# B&R Automation Studio project Nitto (part 5)

#### CSV_ReadFile.ab
```automation-basic
FUNCTION_BLOCK CSV_ReadFile
;*****************************************************************
;FUB: 			CSV_ReadFile
;*****************************************************************
;Discription:
;	This FUB reads the Values from a CSV-File.
;
;Parameter:
;
;Author:	Georg Kreil
;			B&R Eggelsberg
;
;History:	V0.01 - 23 June 2003
;					created
;			V0.01.1 - 4 July 2003
;					no changes
;			V0.01.2 - 8 July 2003
;					Error with array-structures corrected
;			V0.01.3 - 14 July 2003
;					Error with array-structures corrected
;			V0.01.4 - 15 July 2003
;					Error by empty rows corrected
;			V0.01.5 - 17 July 2003
;					Error, when variable starts with array-structure, corrected
;			V0.01.6 - 21 July 2003
;					strings can have all possible character without ";"
;			V0.01.7 - 7 August 2003
;					no changes
;			V0.01.8 - 8 August 2003
;					no changes
;			V0.01.9 - 11 August 2003
;					Value error corrected
;			V0.02.0
;					no changes
;			V0.02.1
;					no changes
;			V0.02.2 - 11 August 2003
;					Datatypcontrol enable/disable
;			V0.02.3
;					no changes
;			V0.02.4 - 4 November 2003
;					Datatyperror in loop corrected
;			V0.02.5 - 13 November 2003
;					Real values error corrected (5e-7)
;			V0.02.6 - 14 November 2003
;					dynamic varible now possible
;			V0.02.7 - 24 November 2003
;					bugfixes
;			V0.02.8 - 27 November 2003
;					changing 80 characters per cyclic to one row per cyclic
;					different bugfixes
;			V0.03.1 - 21 January 2004
;					using the created strings from FUB CSV_ListFile with date
;			V0.03.3 - 12 May 2004
;					array behind array-structure corrected
;			V0.03.4 - 14 May 2004
;					changed the UDINT-conversion from STRING (see CSV_SEARCH)
;					corrected the STRING-datatypcontrol (1Byte error)
;			V0.03.9 - 2 August 2004
;					correction "only array" and "only array in struct"
;
;*****************************************************************
temp_status = temp_status
Options = Options

Internal.CharPerCyclic= 80		; number of character

loop Internal.y=0 to 10 do
	select Internal.Step

		;##########################################################################################
		state WAIT
		;##########################################################################################

			Internal.FileIdent= 0
			Internal.temp_status=0
			VarCnt = 0
			Internal.Separator = Separator

			if( (Internal.Separator = '.') or (Internal.Separator = '[') or (Internal.Separator = ']') or (Internal.Separator <= 32) or ( (Internal.Separator >= '0') and (Internal.Separator <= '9') ) or ( (Internal.Separator >= 'a') and (Internal.Separator <= 'z') ) or ( (Internal.Separator >= 'A') and (Internal.Separator <= 'Z') ) ) then
				status = ERROR_WRONG_SEPARATOR
				exitif(1=1)
			endif

			strcpy(adr(Internal.FileName),pFileName)
			if (Internal.y=0) then
				if( strlen(adr(Internal.FileName)) <> 0 ) then
					; control, if the filename has the right extension
					loop Internal.i=0 to sizeof(Internal.FileName) do

						Dyn_Usint access (adr(Internal.FileName)+Internal.i)

						; this is for using the created strings from FUB CSV_ListFile
						if (Dyn_Usint = ' ') then
							Dyn_Usint= 0
							; add extension to filename
							strcpy((adr(Internal.FileName)+Internal.i),".CSV")
							exitif(1=1)
						endif

						if(Dyn_Usint = '.')then
							if ( strcmp((adr(Internal.FileName)+Internal.i),".CSV") = 0 ) or ( strcmp((adr(Internal.FileName)+Internal.i),".csv") = 0 ) then
								exitif(1=1)
							else
								; replace wrong extension
								strcpy((adr(Internal.FileName)+Internal.i),".CSV")
								exitif(1=1)
							endif
						else if(Dyn_Usint = 0) then
							; add extension to filename
							strcpy((adr(Internal.FileName)+Internal.i),".CSV")
							exitif(1=1)
						endif

					endloop
					Internal.ArrayStructureStarts= 0
					status= 65535
					;Pathname angegeben
					if(pPath <> 0)then
						strcpy(adr(Internal.Path),pPath)
						; Pathname bearbeiten
						if( strlen(adr(Internal.Path)) <> 0 )then

						; control, if the filename has the right extension
							loop Internal.i=0 to sizeof(Internal.Path) do

								Dyn_Usint access (adr(Internal.Path) + Internal.i)
								 if( ((Dyn_Usint >= '0' ) and ( Dyn_Usint <= '9' )) or ((Dyn_Usint >= 'A') and (Dyn_Usint <= 'Z')) or ((Dyn_Usint >= 'a') and (Dyn_Usint <= 'z')) or ( Dyn_Usint = '_') or ( Dyn_Usint = '-') or ( Dyn_Usint = '/') or ( Dyn_Usint = '\') or ( Dyn_Usint = 0) )then

									if(Dyn_Usint = 0) then
										Dyn_Usint access (adr(Internal.Path) + Internal.i - 1)
										if(Dyn_Usint <> '\') and (Dyn_Usint <> '/')then
											strcat( adr(Internal.Path), adr("/") )
										endif
										exitif(1=1)
									endif
									status= 65535
								else
									status= INVALID_CHARACTER
									exitif(1=1)
								endif
							endloop
							strcat( adr(Internal.Path), adr(Internal.FileName) )
							strcpy( adr(Internal.FileName), adr(Internal.Path) )
						endif
					endif

				else
					status= NO_FILENAME
				endif
			endif

			when (1=1) and (Internal.y=0) do
			next FILE_OPEN

		;##########################################################################################
		state FILE_OPEN
		;##########################################################################################

			FileOpen_CSV.enable= 1
			FileOpen_CSV.pDevice= pDevice
			FileOpen_CSV.pFile= adr(Internal.FileName)
			FileOpen_CSV.mode= 2	;FILE_RW
			FileOpen_CSV FUB FileOpen()

			; no error
			when (FileOpen_CSV.status = 0) do
				Internal.FileIdent= FileOpen_CSV.ident
				; allocate memory, to copy the whole file
				Internal.status_alloc= TMP_alloc(FileOpen_CSV.filelen,adr(Internal.pFileData))
				strcpy(adr(Internal.FileName),"")
				status= 65535
			next FILE_READ

			; file is opening
			when (FileOpen_CSV.status = 65535) do
				status= FileOpen_CSV.status
			next FILE_OPEN

			;error durring
			when (FileOpen_CSV.status <> 0) and (FileOpen_CSV.status <> 65535) do
				status= FileOpen_CSV.status
			next WAIT

		;##########################################################################################
		state FILE_READ
		;##########################################################################################

			if( (Internal.status_alloc = 0) and (FileOpen_CSV.status = 0) )then
				FileRead_CSV.enable= 1
				FileRead_CSV.ident= Internal.FileIdent
				FileRead_CSV.offset= 0
				FileRead_CSV.pDest= Internal.pFileData
				FileRead_CSV.len= FileOpen_CSV.filelen
				FileRead_CSV FUB FileRead()
			endif

			when  (Internal.status_alloc <> 0) do
				status= Internal.status_alloc
			next WAIT

			when (FileRead_CSV.status <> 0) and  (FileRead_CSV.status <> 65535) do
				status= FileRead_CSV.status
			next WAIT

			when (FileRead_CSV.status = 65535) do
				status= FileRead_CSV.status
			next FILE_READ

			when (FileRead_CSV.status = 0) do
				Internal.Offset= 0
				Internal.OffsetOld= 0
				Internal.i= 0
				strcpy(adr(Internal.Value),"")
				strcpy(adr(Internal.TmpName),"")
				strcpy(adr(Internal.StructName),"")
				strcpy(adr(Internal.DataTyp),"")
				strcpy(adr(Internal.DateTime),"")
				strcpy(adr(Internal.VarName),"")
				Internal.OnlyArray= 0
				Internal.OnlyArrayInStruct= 0
				LineCnt= 0
				status= 65535
				ErrorNumber = 0
				ErrorLine = 0
				ErrorCnt = 0
			next FILE_CLOSE

		;##########################################################################################
		state FILE_CLOSE
		;##########################################################################################

		 	FileClose_CSV.enable= 1
			FileClose_CSV.ident= Internal.FileIdent
			FileClose_CSV FUB FileClose()

			; Fehler beim Schliessen
			when (FileClose_CSV.status <> 0) and (FileClose_CSV.status <> 65535) do
				status= FileClose_CSV.status
			next WAIT

			; kein Fehler aufgetreten
			when (FileClose_CSV.status = 0) do
				status= 65535
			next SEARCH_STRUCT_NAME

			; noch nicht fertig
			when (FileClose_CSV.status = 65535) do
				status= FileClose_CSV.status
			next FILE_CLOSE

		;##########################################################################################
		state SEARCH_STRUCT_NAME
		;##########################################################################################

		when (Internal.Offset >= FileOpen_CSV.filelen) or (status <> 65535) do
		next TEMP_FREE

		loop
			SearchChar access Internal.pFileData + Internal.Offset
			TestUsint = SearchChar

			if( SearchChar = 13 )then
				LineCnt= LineCnt+1
			endif

			if( SearchChar = '/' ) and (Internal.NameEntered <> 2) then
				Internal.HeaderLine= 1
			; date and time
			else if( (((SearchChar >= '0' ) and ( SearchChar <= '9' )) or ((SearchChar >= 'A') and (SearchChar <= 'Z')) or ((SearchChar >= 'a') and (SearchChar <= 'z')) or ( SearchChar = '.') or (SearchChar = ':') or (SearchChar = ' ') ) and (strcmp(adr(Internal.DataTyp),"DATE_AND_TIME") = 0 ) and (Internal.NameEntered = 2) and (Internal.HeaderLine = 0) )then			; neue Zeile
				Internal.DateTime[Internal.j]= SearchChar
				Internal.j= Internal.j+1
				Internal.DateAndTime= 1
			; only numbers
			else if( (((SearchChar >= '0' ) and ( SearchChar <= '9' )) or ( SearchChar = '.')  or ( SearchChar = 'E') or ( SearchChar = 'e') or ( SearchChar = '-')) and (Internal.NameEntered = 2) and (Internal.HeaderLine = 0) )then			; neue Zeile
				Internal.Value[Internal.j]= SearchChar
				Internal.j= Internal.j+1
			; Strings
	;		else if( (((SearchChar >= '0' ) and ( SearchChar <= '9' )) or ((SearchChar >= 'A') and (SearchChar <= 'Z')) or((SearchChar >= 'a') and (SearchChar <= 'z'))  or ( SearchChar = '.') or ( SearchChar = ' ')) and (Internal.NameEntered = 2) and (strcmp(adr(Internal.DataTyp),"STRING") = 0) and (Internal.HeaderLine = 0) )then			; neue Zeile
	;		else if( (((SearchChar >= 33 ) and ( SearchChar <= 58 )) or ((SearchChar >= 60 ) and ( SearchChar <= 126 )) or ( SearchChar = ' ') ) and (Internal.NameEntered = 2) and (strcmp(adr(Internal.DataTyp),"STRING") = 0) and (Internal.HeaderLine = 0) )then			; neue Zeile
;			alle sinnvollen Zeichen zulassen, auch Sonderzeichen
			else if( (SearchChar >= 32 ) and ( SearchChar <= 126 ) and (Internal.NameEntered = 2) and (strcmp(adr(Internal.DataTyp),"STRING") = 0) and (Internal.HeaderLine = 0) )then			; neue Zeile
				Internal.Value[Internal.j]= SearchChar
				Internal.j= Internal.j+1
			else if( ((SearchChar >= 'A') and (SearchChar <= 'Z')) or ((SearchChar >= 'a') and (SearchChar <= 'z')) or ((SearchChar >= '0' ) and ( SearchChar <= '9' )) or (SearchChar = '.') or (SearchChar = ':') or (SearchChar = '*') or (SearchChar = '[') or (SearchChar = ']') or (SearchChar = '_') and (Internal.HeaderLine = 0) )then
				Internal.TmpName[Internal.i]= SearchChar
				Internal.i= Internal.i+1
			else if( SearchChar = 13 ) or ( SearchChar = 10 )  then			; neue Zeile
				SearchChar access Internal.pFileData + Internal.Offset+1
				TestUsint = SearchChar
				if( SearchChar = 10) or ( SearchChar = 13 ) then
	;				LineCnt= LineCnt+1
					if(Internal.NameEntered = 1) then
						Internal.TmpName[Internal.i]= 0
						Internal.i= 0
						strcpy(adr(Internal.DataTyp),adr(Internal.TmpName))
					endif
					Internal.Value[Internal.j]= 0
					Internal.DateTime[Internal.j]= 0
					Internal.i= 0
					Internal.j= 0
					Internal.TmpName[Internal.i]= 0
					Internal.NameEntered= 0
					Internal.HeaderLine= 0
					inc(Internal.Offset)
					exitif(strlen(adr(Internal.StructName)) <> 0)
	;				exitif(1=1)
				else
	;				LineCnt= LineCnt+1
					if(Internal.NameEntered = 1) then
						Internal.TmpName[Internal.i]= 0
						Internal.i= 0
						strcpy(adr(Internal.DataTyp),adr(Internal.TmpName))
					endif
					Internal.Value[Internal.j]= 0
					Internal.DateTime[Internal.j]= 0
					Internal.i= 0
					Internal.j= 0
					Internal.TmpName[Internal.i]= 0
					Internal.NameEntered= 0
					Internal.HeaderLine= 0
					exitif(strlen(adr(Internal.StructName)) <> 0)
	;				exitif(1=1)
				endif
			; the structure name was readed
			else if( SearchChar = Internal.Separator) and (Internal.NameEntered = 0) and (Internal.HeaderLine = 0) then		; neuer Name
				Internal.TmpName[Internal.i]= 0
				Internal.i= 0
				strcpy(adr(Internal.StructName),adr(Internal.TmpName))
				Internal.NameEntered= 1
			; dataype was readed
			else if( SearchChar = Internal.Separator) and (Internal.NameEntered = 1) and (Internal.HeaderLine = 0) then		; neuer Datentyp
				Internal.TmpName[Internal.i]= 0
				Internal.i= 0
				strcpy(adr(Internal.DataTyp),adr(Internal.TmpName))
				Internal.NameEntered= 2
			; value was readed
			else if( SearchChar = Internal.Separator) and (Internal.NameEntered = 2) and (Internal.HeaderLine = 0) then		; weitere Spalten ignorieren
				Internal.TmpName[Internal.j]= 0
				Internal.NameEntered= 3

			else if( SearchChar = ' ') and (Internal.NameEntered = 0) and (Internal.HeaderLine = 0) then		; Leerzeichen
				Internal.SpacesCounter= Internal.SpacesCounter+1
			endif
			exitif(Internal.Offset >= FileOpen_CSV.filelen+1)
			inc(Internal.Offset)
		endloop

		Internal.Offset= Internal.Offset+1
		Internal.OffsetOld= Internal.Offset
		memcpy(adr(Internal.TmpDataTyp),adr(Internal.DataTyp),5)
		Internal.TmpDataTyp[5]= 0

;		when (RowNotOnEnd = 1) do
;			status= 65535
;		next SEARCH_STRUCT_NAME

		; is it a dynamic variable
		if(Internal.StructName[0] = '*')then
			Internal.DynamicVariable= 1
		else
			Internal.DynamicVariable= 0
		endif

		;######################################################
		; Correction 15.July 2003
		when ( strlen(adr(Internal.StructName)) = 0  )do
			status= 65535
		next SEARCH_STRUCT_NAME
		; Correction 15.July 2003
		;######################################################

		when (Internal.HeaderLine = 1)do
			status= 65535
		next SEARCH_STRUCT_NAME

		;######################################################
		; Correction 17.July 2003
		when( strcmp(adr(Internal.DataTyp),"ARRAY_OF_STRUCTURES") = 0 ) do
			loop Internal.i=strlen(adr(Internal.StructName)) downto 0 do	;Kommastellen löschen
				SearchChar access adr(Internal.StructName)+Internal.i
				if(SearchChar ='.')then
					SearchChar= 0
					Part=1
					exitif(1=1)
				endif
			endloop
			if(	Part = 0 )then
				Internal.ArrayStructureStarts= 1
				strcpy(adr(Internal.StructName),"")
				Internal.i= 0
				Internal.SpacesCounter= 0
			else
				strcat(adr(Internal.StructName),adr(Internal.VarName))
				Internal.i= 0
				Internal.SpacesCounter= 0
				Part= 0
				status= 65535
			endif
		next SEARCH_VAR_NAMES

	;	when( ( strcmp(adr(Internal.DataTyp),"STRUCTURE") = 0 ) or ( strcmp(adr(Internal.DataTyp),"ARRAY_OF_STRUCTURES") = 0 ) ) do
		when ( strcmp(adr(Internal.DataTyp),"STRUCTURE") = 0 ) do
		; Correction 17.July 2003
		;######################################################
			Internal.level= 2
			loop Internal.i=0 to strlen(adr(Internal.StructName)) do
				SearchChar access adr(Internal.StructName)+Internal.i
				if(SearchChar ='.') and( Internal.level = ((Internal.SpacesCounter+1)/5) ) then
					SearchChar= 0
					exitif(1=1)
				else if(SearchChar =']') and( Internal.level = ((Internal.SpacesCounter+1)/5) ) then
					SearchChar access adr(Internal.StructName)+Internal.Merker
					SearchChar= 0
					exitif(1=1)
				else if (SearchChar ='.') and ( Internal.level < ((Internal.SpacesCounter+1)/5) ) then
					Internal.level= Internal.level+1
				else if (SearchChar =']') and ( Internal.level < ((Internal.SpacesCounter+1)/5) ) then
					Internal.level= Internal.level+1
				endif
			endloop
			Internal.i=0

			strcat(adr(Internal.StructName),adr(Internal.VarName))

			Internal.SpacesCounter= 0
			status= 65535
		next SEARCH_VAR_NAMES

		when(strcmp(adr(Internal.TmpDataTyp),"ARRAY") = 0 ) do
			Internal.OnlyArray= 1
			loop Internal.i=strlen(adr(Internal.StructName)) downto 0 do
				SearchChar access adr(Internal.StructName) + Internal.i
				if(SearchChar ='.')then
					SearchChar = 0
					Internal.OnlyArray= 0
					Internal.OnlyArrayInStruct= 1
					exitif(1=1)
				endif
			endloop

			Internal.i=0
			status= 65535
		next SEARCH_VAR_NAMES

		when( 1=1 ) do
			Internal.level= 2
			loop Internal.i=0 to strlen(adr(Internal.StructName)) do
				SearchChar access adr(Internal.StructName)+Internal.i
				if(SearchChar ='.') and( Internal.level = ((Internal.SpacesCounter+1)/5) ) then
					SearchChar= 0
					exitif(1=1)
				else if(SearchChar =']') and( Internal.level = ((Internal.SpacesCounter+1)/5) ) then
					SearchChar access adr(Internal.StructName)+Internal.Merker
					SearchChar= 0
					exitif(1=1)
				else if (SearchChar ='.') and ( Internal.level < ((Internal.SpacesCounter+1)/5) ) then
					Internal.level= Internal.level+1
				else if (SearchChar =']') and ( Internal.level < ((Internal.SpacesCounter+1)/5) ) then
					Internal.level= Internal.level+1
				endif
			endloop
			Internal.i=0
			strcat(adr(Internal.StructName),adr(Internal.VarName))

			Internal.SpacesCounter= 0
			status= 65535
		next SET_VARIABLE

		;##########################################################################################
		state SEARCH_VAR_NAMES
		;##########################################################################################

		when (Internal.Offset >= FileOpen_CSV.filelen) or (status <> 65535) do
		next TEMP_FREE

		loop
			SearchChar access Internal.pFileData + Internal.Offset
			TestUsint = SearchChar

			if( LineCnt = 64 )then
				LineCnt = LineCnt
			endif

			if( SearchChar = 13 )then
				LineCnt= LineCnt+1
			endif

			if( SearchChar = '/' ) and (Internal.NameEntered <> 2) then
				Internal.HeaderLine= 1
			; Zeit/Datum
			else if( (((SearchChar >= '0' ) and ( SearchChar <= '9' )) or ((SearchChar >= 'A') and (SearchChar <= 'Z')) or ((SearchChar >= 'a') and (SearchChar <= 'z')) or ( SearchChar = '.') or (SearchChar = ':') or (SearchChar = ' ') ) and (strcmp(adr(Internal.DataTyp),"DATE_AND_TIME") = 0 ) and (Internal.NameEntered = 2) and (Internal.HeaderLine = 0)  )then			; neue Zeile
				Internal.DateTime[Internal.j]= SearchChar
				Internal.j= Internal.j+1
			; Nur Zahlenwert
			else if( (((SearchChar >= '0' ) and ( SearchChar <= '9' )) or ( SearchChar = '.')  or ( SearchChar = 'E') or ( SearchChar = 'e') or ( SearchChar = '-')) and (Internal.NameEntered = 2) and (Internal.HeaderLine = 0) )then			; neue Zeile
				Internal.Value[Internal.j]= SearchChar
				Internal.j= Internal.j+1
			; String-Wert
	;		else if( (((SearchChar >= '0' ) and ( SearchChar <= '9' )) or ((SearchChar >= 'A') and (SearchChar <= 'Z')) or((SearchChar >= 'a') and (SearchChar <= 'z'))  or ( SearchChar = '.') or ( SearchChar = ' ')) and (Internal.NameEntered = 2) and (strcmp(adr(Internal.DataTyp),"STRING") = 0) and (Internal.HeaderLine = 0) )then			; neue Zeile
;			else if( (((SearchChar >= 33 ) and ( SearchChar <= 58 )) or ((SearchChar >= 60 ) and ( SearchChar <= 126 )) or ( SearchChar = ' ') ) and (Internal.NameEntered = 2) and (strcmp(adr(Internal.DataTyp),"STRING") = 0) and (Internal.HeaderLine = 0) )then			; neue Zeile
;			alle sinnvollen Zeichen zulassen, auch Sonderzeichen
			else if( (SearchChar >= 32 ) and ( SearchChar <= 126 ) and (Internal.NameEntered = 2) and (strcmp(adr(Internal.DataTyp),"STRING") = 0) and (Internal.HeaderLine = 0) )then			; neue Zeile
				Internal.Value[Internal.j]= SearchChar
				Internal.j= Internal.j+1
			else if( ((SearchChar >= 'A') and (SearchChar <= 'Z')) or ((SearchChar >= 'a') and (SearchChar <= 'z')) or ((SearchChar >= '0' ) and ( SearchChar <= '9' )) or (SearchChar = '.') or (SearchChar = ':') or (SearchChar = '*') or (SearchChar = '[') or (SearchChar = ']') or (SearchChar = '_') and (Internal.HeaderLine = 0) )then
				Internal.TmpName[Internal.i]= SearchChar
				Internal.i= Internal.i+1
			else if( SearchChar = 13 ) or ( SearchChar = 10 )  then			; neue Zeile
				Internal.Offset= Internal.Offset+1
	;			LineCnt= LineCnt+1
				SearchChar access Internal.pFileData + Internal.Offset
				TestUsint = SearchChar
				if( SearchChar = 10) or ( SearchChar = 13 ) then
	;				LineCnt= LineCnt+1
					if(Internal.NameEntered = 1) then
						Internal.TmpName[Internal.i]= 0
						Internal.i= 0
						strcpy(adr(Internal.DataTyp),adr(Internal.TmpName))
					endif
					Internal.Value[Internal.j]= 0
					Internal.DateTime[Internal.j]= 0
					Internal.i= 0
					Internal.j= 0
					Internal.TmpName[Internal.i]= 0
					Internal.NameEntered= 0
					inc(Internal.Offset)
;					Internal.HeaderLine= 0
					exitif( (strlen(adr(Internal.VarName)) <> 0) or (Internal.HeaderLine= 1) )
				else
	;				LineCnt= LineCnt+1
					if(Internal.NameEntered = 1) then
						Internal.TmpName[Internal.i]= 0
						Internal.i= 0
						strcpy(adr(Internal.DataTyp),adr(Internal.TmpName))
					endif
					if(strlen(adr(Internal.VarName)) = 0) then
						Internal.Offset= Internal.Offset-1
					endif
					Internal.Value[Internal.j]= 0
					Internal.DateTime[Internal.j]= 0
					Internal.i= 0
					Internal.j= 0
					Internal.TmpName[Internal.i]= 0
					Internal.NameEntered= 0
;					Internal.HeaderLine= 0
					exitif( (strlen(adr(Internal.VarName)) <> 0) or (Internal.HeaderLine= 1) )
				endif
			; Strukturname
			else if( SearchChar = Internal.Separator) and (Internal.NameEntered = 0) and (Internal.HeaderLine = 0) then		; neuer Name
				Internal.TmpName[Internal.i]= 0
				Internal.i= 0
				Internal.j= 0			; Correction 11 August 2003
				strcpy(adr(Internal.VarName),adr(Internal.TmpName))
				Internal.NameEntered= 1
			; Datenyp
			else if( SearchChar = Internal.Separator) and (Internal.NameEntered = 1) and (Internal.HeaderLine = 0) then		; neuer Datentyp
				Internal.TmpName[Internal.i]= 0
				Internal.i= 0
				Internal.j= 0			; Correction 11 August 2003
				strcpy(adr(Internal.DataTyp),adr(Internal.TmpName))
				Internal.NameEntered= 2

			else if( SearchChar = Internal.Separator) and (Internal.NameEntered = 2) and (Internal.HeaderLine = 0) then		; weitere Spalten ignorieren
				Internal.TmpName[Internal.j]= 0
				Internal.NameEntered= 3

			else if( SearchChar = ' ') and (Internal.NameEntered = 0) and (Internal.HeaderLine = 0) then		; Leerzeichen
				Internal.SpacesCounter= Internal.SpacesCounter+1
			endif
			exitif(Internal.Offset >= FileOpen_CSV.filelen+1)
			inc(Internal.Offset)
		endloop

	;	Internal.Offset= Internal.Offset+1
			Internal.Offset= Internal.Offset
		Internal.OffsetOld= Internal.Offset
		memcpy(adr(Internal.TmpDataTyp),adr(Internal.DataTyp),5)
		Internal.TmpDataTyp[5]= 0

;		when (RowNotOnEnd = 1) do
;			status= 65535
;		next SEARCH_VAR_NAMES

		when (Internal.HeaderLine = 1)do
			Internal.HeaderLine = 0
			Internal.i= 0
			strcpy(adr(Internal.Value),"")
			strcpy(adr(Internal.TmpName),"")
			strcpy(adr(Internal.StructName),"")
			strcpy(adr(Internal.DataTyp),"")
			strcpy(adr(Internal.DateTime),"")
			strcpy(adr(Internal.VarName),"")
			Internal.OnlyArray= 0
			Internal.OnlyArrayInStruct= 0
			Internal.ArrayStructureStarts = 0
			status= 65535
		next SEARCH_STRUCT_NAME

		;######################################################
		; Correction 6.October 2003
		when ( strlen(adr(Internal.StructName)) = 0  )and (Internal.ArrayStructureStarts = 0) do
			status= 65535
		next SEARCH_STRUCT_NAME
		; Correction 6.October 2003
		;######################################################

		;no new variablename in csv-file found
		when (Internal.VarName[0] = 0) do
			Internal.StructName[0]= 0
			status= 65535
		next SEARCH_STRUCT_NAME

		; full name found
		when(Internal.VarName[0]<> '.') do
			strcpy(adr(Internal.StructName),adr(Internal.VarName))
			status= 65535
		next SET_VARIABLE

		; only array-variable -> no structure, no single variable
		when(Internal.OnlyArray = 1) do
			; is it a dynamic variable
			if(Internal.DynamicVariable = 1)then
				strcat( adr(Internal.StructName), "*" )
				strcat( adr(Internal.StructName), adr(Internal.VarName)+1)
			else
				strcpy( adr(Internal.StructName), adr(Internal.VarName)+1)
			endif

			status= 65535
		next SET_VARIABLE

		; only an array-variable in a structure -> no structure, no single variable
		when(Internal.OnlyArrayInStruct = 1) do
			Internal.i=0
			strcat( adr(Internal.StructName), adr(Internal.VarName))
			status= 65535
		next SET_VARIABLE

		; beginn of an array of structures found
		when( strcmp(adr(Internal.DataTyp),"ARRAY_OF_STRUCTURES") = 0 ) do

			Internal.level= 2
			loop Internal.i=0 to strlen(adr(Internal.StructName)) do
				SearchChar access adr(Internal.StructName)+Internal.i
				if(SearchChar ='.') and( Internal.level = ((Internal.SpacesCounter+1)/5) ) then
					SearchChar= 0
					exitif(1=1)
				else if(SearchChar =']') and( Internal.level = ((Internal.SpacesCounter+1)/5) ) then
					SearchChar access adr(Internal.StructName)+Internal.Merker
					SearchChar= 0
					exitif(1=1)
				else if (SearchChar ='.') and ( Internal.level < ((Internal.SpacesCounter+1)/5) ) then
					Internal.level= Internal.level+1
				else if (SearchChar =']') and ( Internal.level < ((Internal.SpacesCounter+1)/5) ) then
					Internal.level= Internal.level+1
				endif
			endloop
			Internal.i=0
			Internal.SpacesCounter= 0
			status= 65535
		next SEARCH_VAR_NAMES

		;new array found
		when ( strcmp(adr(Internal.TmpDataTyp),"ARRAY") = 0 )do
			Internal.level= 2
			loop Internal.i=0 to strlen(adr(Internal.StructName)) do
				SearchChar access adr(Internal.StructName)+Internal.i
				if(SearchChar ='.') and( Internal.level = ((Internal.SpacesCounter+1)/5) ) then
					SearchChar= 0
					exitif(1=1)
				else if(SearchChar =']') and( Internal.level = ((Internal.SpacesCounter+1)/5) ) then
					SearchChar access adr(Internal.StructName)+Internal.Merker
					SearchChar= 0
					exitif(1=1)
				else if (SearchChar ='.') and ( Internal.level < ((Internal.SpacesCounter+1)/5) ) then
					Internal.level= Internal.level+1
				else if (SearchChar =']') and ( Internal.level < ((Internal.SpacesCounter+1)/5) ) then
					Internal.level= Internal.level+1
				endif
			endloop
			Internal.i=0
			Internal.SpacesLastRow= Internal.SpacesCounter
			Internal.SpacesCounter= 0
			status= 65535
		next SEARCH_VAR_NAMES

		; new structure found
		when( strcmp(adr(Internal.DataTyp),"STRUCTURE") = 0 ) do
		;######################################################
		; Correction 17.July 2003
			if (Internal.ArrayStructureStarts = 0) then
				Internal.level= 2
				loop Internal.i=0 to strlen(adr(Internal.StructName)) do
					SearchChar access adr(Internal.StructName)+Internal.i
					if(SearchChar ='.') and( Internal.level = ((Internal.SpacesCounter+1)/5) ) then
						SearchChar= 0
						exitif(1=1)
					else if(SearchChar =']') and( Internal.level = ((Internal.SpacesCounter+1)/5) ) then

						loop Internal.j=Internal.i downto 0 do
							SearchChar access adr(Internal.StructName)+Internal.j
							exitif(SearchChar = '.')
						endloop
						SearchChar= 0
						exitif(1=1)
					else if (SearchChar ='.') and ( Internal.level < ((Internal.SpacesCounter+1)/5) ) then
						Internal.level= Internal.level+1
					else if (SearchChar =']') and ( Internal.level < ((Internal.SpacesCounter+1)/5) ) then
						Internal.level= Internal.level+1
					endif
				endloop
				Internal.i=0
				strcat(adr(Internal.StructName),adr(Internal.VarName))
			else
				Internal.level= 2
				if(( Internal.level <> ((Internal.SpacesCounter+1)/5) )) then
					loop Internal.i=0 to strlen(adr(Internal.StructName)) do
						SearchChar access adr(Internal.StructName)+Internal.i
						if(SearchChar ='.') and( Internal.level = ((Internal.SpacesCounter+1)/5) ) then
							SearchChar= 0
							exitif(1=1)
						else if(SearchChar =']') and( Internal.level = ((Internal.SpacesCounter+1)/5) ) then

							loop Internal.j=Internal.i downto 0 do
								SearchChar access adr(Internal.StructName)+Internal.j
								exitif(SearchChar = '.')
							endloop
							SearchChar= 0
							exitif(1=1)
						else if (SearchChar ='.') and ( Internal.level < ((Internal.SpacesCounter+1)/5) ) then
							Internal.level= Internal.level+1
						else if (SearchChar =']') and ( Internal.level < ((Internal.SpacesCounter+1)/5) ) then
							Internal.level= Internal.level+1
						endif
					endloop
				else
					Internal.i= 0
					; is it a dynamic variable
					if(Internal.DynamicVariable = 1)then
						strcpy( adr(Internal.StructName),"*" )
					else
						strcpy( adr(Internal.StructName),"" )
					endif
				endif

				if ( Internal.i = 0 ) then
					strcat(adr(Internal.StructName),adr(Internal.VarName)+1)
				else
					strcat(adr(Internal.StructName),adr(Internal.VarName))
				endif
				Internal.i=0
			endif
		; Correction 17.July 2003
		;######################################################

			Internal.SpacesCounter= 0
			status= 65535
		next SEARCH_VAR_NAMES

		when( 1=1 ) do
			Internal.level= 2
			loop Internal.i=0 to strlen(adr(Internal.StructName)) do
				SearchChar access adr(Internal.StructName)+Internal.i
				if(SearchChar ='.') and( Internal.level = ((Internal.SpacesCounter+1)/5) ) then
					SearchChar= 0
					exitif(1=1)
				else if(SearchChar =']') and( Internal.level = ((Internal.SpacesCounter+1)/5) ) then
					SearchChar access adr(Internal.StructName)+Internal.Merker
					SearchChar= 0
					exitif(1=1)
				else if (SearchChar ='.') and ( Internal.level < ((Internal.SpacesCounter+1)/5) ) then
					Internal.Merker= Internal.i
					Internal.level= Internal.level+1
				else if (SearchChar =']') and ( Internal.level < ((Internal.SpacesCounter+1)/5) ) then
					Internal.level= Internal.level+1
				endif
			endloop
			Internal.i=0
			strcat(adr(Internal.StructName),adr(Internal.VarName))

			Internal.SpacesCounter= 0
			status= 65535
		next SET_VARIABLE

		;##########################################################################################
		state SET_VARIABLE
		;##########################################################################################

		Internal.PV_xgetadrStatus= PV_xgetadr(adr(Internal.StructName), adr(Internal.PV_Adress), adr(Internal.data_len))
		Internal.PV_nInfoStatus= PV_ninfo(adr(Internal.StructName),adr(Internal.PVdata_typ),adr(Internal.datatyp_len),adr(Internal.dimension))

		when(	Internal.PV_xgetadrStatus <> 0 ) and (IgnoreError = FALSE) do
			Internal.OnlyArrayInStruct = 0
			if( ErrorNumber = 0 ) then
				ErrorNumber = Internal.PV_xgetadrStatus
				ErrorLine = LineCnt
			endif

			inc( ErrorCnt )
			status= Internal.PV_xgetadrStatus
		next TEMP_FREE

		when(	Internal.PV_xgetadrStatus <> 0 ) and (IgnoreError = TRUE) do
			if( ErrorNumber = 0 ) then
				ErrorNumber = Internal.PV_xgetadrStatus
				ErrorLine = LineCnt
			endif

			inc( ErrorCnt )

			status= 65535
		next SEARCH_VAR_NAMES

		Inc(VarCnt)

		if( (strcmp(adr(Internal.DataTyp),"BOOL") = 0 ) and (Internal.data_len = 1) and (Internal.PV_xgetadrStatus = 0) and (Internal.PV_nInfoStatus = 0) )then

			if (Internal.PVdata_typ = 1) then
				Dyn_Bool access Internal.PV_Adress
				loop Internal.i=strlen(adr(Internal.Value)) downto 0 do	;Kommastellen löschen
					SearchChar access adr(Internal.Value)+Internal.i
					if(SearchChar ='.')then
						SearchChar= 0
						exitif(1=1)
					endif
				endloop
				Dyn_Bool= bool( atoi(adr(Internal.Value)) )
				status= 65535
			else
				Internal.OnlyArrayInStruct = 0
				Internal.temp_status= DATATYP_ERROR
			endif

		else if( (strcmp(adr(Internal.DataTyp),"USINT") = 0 ) and (Internal.data_len = 1) and (Internal.PV_xgetadrStatus = 0) and (Internal.PV_nInfoStatus = 0) )then

			if (Internal.PVdata_typ = 5) then
				Dyn_Usint access Internal.PV_Adress
				loop Internal.i=strlen(adr(Internal.Value)) downto 0 do	;Kommastellen löschen
					SearchChar access adr(Internal.Value)+Internal.i
					if(SearchChar ='.')then
						SearchChar= 0
						exitif(1=1)
					endif
				endloop
				Dyn_Usint= usint( atoi(adr(Internal.Value)) )
				status= 65535
			else
				Internal.OnlyArrayInStruct = 0
				Internal.temp_status= DATATYP_ERROR
			endif

		else if( (strcmp(adr(Internal.DataTyp),"SINT") = 0 ) and (Internal.data_len = 1) and (Internal.PV_xgetadrStatus = 0) and (Internal.PV_nInfoStatus = 0) )then

			if (Internal.PVdata_typ = 2) then
				Dyn_Sint access Internal.PV_Adress
				loop Internal.i=strlen(adr(Internal.Value)) downto 0 do	;Kommastellen löschen
					SearchChar access adr(Internal.Value)+Internal.i
					if(SearchChar ='.')then
						SearchChar= 0
						exitif(1=1)
					endif
				endloop
				Dyn_Sint= sint( atoi(adr(Internal.Value)) )
				status= 65535
			else
				Internal.OnlyArrayInStruct = 0
				Internal.temp_status= DATATYP_ERROR
			endif

		else if( (strcmp(adr(Internal.DataTyp),"UINT") = 0 ) and (Internal.data_len = 2) and (Internal.PV_xgetadrStatus = 0) and (Internal.PV_nInfoStatus = 0) )then

			if (Internal.PVdata_typ = 6) then
				Dyn_Uint access Internal.PV_Adress
				loop Internal.i=strlen(adr(Internal.Value)) downto 0 do	;Kommastellen löschen
					SearchChar access adr(Internal.Value)+Internal.i
					if(SearchChar ='.')then
						SearchChar= 0
						exitif(1=1)
					endif
				endloop
				Dyn_Uint= uint( atoi(adr(Internal.Value)) )
				status= 65535
			else
				Internal.OnlyArrayInStruct = 0
				Internal.temp_status= DATATYP_ERROR
			endif

		else if( (strcmp(adr(Internal.DataTyp),"INT") = 0 ) and (Internal.data_len = 2) and (Internal.PV_xgetadrStatus = 0) and (Internal.PV_nInfoStatus = 0) )then

			if (Internal.PVdata_typ = 3) then
				Dyn_Int access Internal.PV_Adress
				loop Internal.i=strlen(adr(Internal.Value)) downto 0 do	;Kommastellen löschen
					SearchChar access adr(Internal.Value)+Internal.i
					if(SearchChar ='.')then
						SearchChar= 0
						exitif(1=1)
					endif
				endloop
				Dyn_Int= int( atoi(adr(Internal.Value)) )
				status= 65535
			else
				Internal.OnlyArrayInStruct = 0
				Internal.temp_status= DATATYP_ERROR
			endif

		else if( (strcmp(adr(Internal.DataTyp),"UDINT") = 0 ) and (Internal.data_len = 4) and (Internal.PV_xgetadrStatus = 0) and (Internal.PV_nInfoStatus = 0) )then

			if (Internal.PVdata_typ = 7) then
				Dyn_Udint access Internal.PV_Adress
				loop Internal.i=strlen(adr(Internal.Value)) downto 0 do	;Kommastellen löschen
					SearchChar access adr(Internal.Value)+Internal.i
					if(SearchChar ='.')then
						SearchChar= 0
						exitif(1=1)
					endif
				endloop

				if (Internal.Value[0] <> '-') then
					Dyn_Udint = 0
					Internal.j = usint(strlen(adr(Internal.Value)))
					loop Internal.i=0 to Internal.j do

						Dyn_Udint = Dyn_Udint+(Internal.Value[Internal.i]-48)*udint(EXPT(10,strlen(adr(Internal.Value))-Internal.i-1))

					endloop
				else
					Dyn_Udint= udint( atoi(adr(Internal.Value)) )
				endif
				status= 65535
			else
				Internal.OnlyArrayInStruct = 0
				Internal.temp_status= DATATYP_ERROR
			endif

		else if( (strcmp(adr(Internal.DataTyp),"DINT") = 0 ) and (Internal.data_len = 4) and (Internal.PV_xgetadrStatus = 0) and (Internal.PV_nInfoStatus = 0) )then

			if (Internal.PVdata_typ = 4) then
				Dyn_Dint access Internal.PV_Adress
				loop Internal.i=strlen(adr(Internal.Value)) downto 0 do	;Kommastellen löschen
					SearchChar access adr(Internal.Value)+Internal.i
					if(SearchChar ='.')then
						SearchChar= 0
						exitif(1=1)
					endif
				endloop
				Dyn_Dint= atoi(adr(Internal.Value))
				status= 65535
			else
				Internal.OnlyArrayInStruct = 0
				Internal.temp_status= DATATYP_ERROR
			endif

		else if( (strcmp(adr(Internal.DataTyp),"STRING") = 0 ) and ((Internal.data_len-1) <= sizeof(Dyn_String)) and ((Internal.data_len-1) >= strlen(adr(Internal.Value))) and (Internal.PV_xgetadrStatus = 0) and (Internal.PV_nInfoStatus = 0) )then

			if (Internal.PVdata_typ = 9) then
				Dyn_String access Internal.PV_Adress
				strcpy(adr(Dyn_String),adr(Internal.Value))
				status= 65535
			else
				Internal.OnlyArrayInStruct = 0
				Internal.temp_status= DATATYP_ERROR
			endif

		else if( (strcmp(adr(Internal.DataTyp),"REAL") = 0 ) and (Internal.data_len = 4) and (Internal.PV_xgetadrStatus = 0) and (Internal.PV_nInfoStatus = 0) )then

			if (Internal.PVdata_typ = 8) then
				Dyn_Real access Internal.PV_Adress
				Dyn_Real= atof(adr(Internal.Value))
				status= 65535
			else
				Internal.OnlyArrayInStruct = 0
				Internal.temp_status= DATATYP_ERROR
			endif

		else if ((strcmp(adr(Internal.DataTyp),"LREAL") = 0 ) and (Internal.data_len = 8) and (Internal.PV_xgetadrStatus = 0) and (Internal.PV_nInfoStatus = 0) )then

			if (Internal.PVdata_typ = 14) then
				Dyn_LReal access Internal.PV_Adress
				Dyn_LReal= CSV_AtoDouble(adr(Internal.Value))
				status= 65535
			else
				Internal.OnlyArrayInStruct = 0
				Internal.temp_status= DATATYP_ERROR
			endif

		else if( (strcmp(adr(Internal.DataTyp),"OCTET STRING") = 0 ) and ((Internal.data_len-1) <= sizeof(Dyn_String)) and ((Internal.data_len-1) >= strlen(adr(Internal.Value))) and (Internal.PV_xgetadrStatus = 0) )then
			Dyn_String access Internal.PV_Adress
			strcpy(adr(Dyn_String),adr(Internal.Value))
			status= 65535

		else if( (strcmp(adr(Internal.DataTyp),"DATE_AND_TIME") = 0 ) and (Internal.data_len = 4) and (Internal.PV_xgetadrStatus = 0) and (Internal.PV_nInfoStatus = 0) )then

			if (Internal.PVdata_typ = 11) then
				Internal.Counter= 0
				loop Internal.i=0 to strlen(adr(Internal.DateTime)) do
					SearchChar access adr(Internal.DateTime)+Internal.i
					if( (SearchChar <> ' ') and (SearchChar <> ':') and (SearchChar <> 0) )then
						Internal.TmpDateTime[Internal.j]= SearchChar
						Internal.j= Internal.j+1
					else if( ((SearchChar = ' ') and (Internal.Counter < 3)) or ((SearchChar = ' ') and (Internal.Counter >= 5)) or ((SearchChar = ':') and (Internal.Counter >= 3)) or (SearchChar = 0) )then
						Internal.TmpDateTime[Internal.j]= 0
						; Tag
						if(Internal.Counter = 0) then
							if(strcmp(adr(Internal.TmpDateTime),"Sun") = 0 )then
								Internal.DateTimeStruct.wday= 0
								Internal.Counter = 1
							else if(strcmp(adr(Internal.TmpDateTime),"Mon") = 0 )then
								Internal.DateTimeStruct.wday= 1
								Internal.Counter = 1
							else if(strcmp(adr(Internal.TmpDateTime),"Tue") = 0 )then
								Internal.DateTimeStruct.wday= 2
								Internal.Counter = 1
							else if(strcmp(adr(Internal.TmpDateTime),"Wed") = 0 )then
								Internal.DateTimeStruct.wday= 3
								Internal.Counter = 1
							else if(strcmp(adr(Internal.TmpDateTime),"Thu") = 0 )then
								Internal.DateTimeStruct.wday= 4
								Internal.Counter = 1
							else if(strcmp(adr(Internal.TmpDateTime),"Fri") = 0 )then
								Internal.DateTimeStruct.wday= 5
								Internal.Counter = 1
							else if(strcmp(adr(Internal.TmpDateTime),"Sat") = 0 )then
								Internal.DateTimeStruct.wday= 6
								Internal.Counter = 1
							endif
						;Datum
						else if(Internal.Counter = 1) then
							if(strcmp(adr(Internal.TmpDateTime),"Jan") = 0 )then
								Internal.DateTimeStruct.month= 1
								Internal.Counter= 2
							else if(strcmp(adr(Internal.TmpDateTime),"Feb") = 0 )then
								Internal.DateTimeStruct.month= 2
								Internal.Counter= 2
							else if(strcmp(adr(Internal.TmpDateTime),"Mar") = 0 )then
								Internal.DateTimeStruct.month= 3
								Internal.Counter= 2
							else if(strcmp(adr(Internal.TmpDateTime),"Apr") = 0 )then
								Internal.DateTimeStruct.month= 4
								Internal.Counter= 2
							else if(strcmp(adr(Internal.TmpDateTime),"May") = 0 )then
								Internal.DateTimeStruct.month= 5
								Internal.Counter= 2
							else if(strcmp(adr(Internal.TmpDateTime),"Jun") = 0 )then
								Internal.DateTimeStruct.month= 6
								Internal.Counter= 2
							else if(strcmp(adr(Internal.TmpDateTime),"Jul") = 0 )then
								Internal.DateTimeStruct.month= 7
								Internal.Counter= 2
							else if(strcmp(adr(Internal.TmpDateTime),"Aug") = 0 )then
								Internal.DateTimeStruct.month= 8
								Internal.Counter= 2
							else if(strcmp(adr(Internal.TmpDateTime),"Sep") = 0 )then
								Internal.DateTimeStruct.month= 9
								Internal.Counter= 2
							else if(strcmp(adr(Internal.TmpDateTime),"Oct") = 0 )then
								Internal.DateTimeStruct.month= 10
								Internal.Counter= 2
							else if(strcmp(adr(Internal.TmpDateTime),"Nov") = 0 )then
								Internal.DateTimeStruct.month= 11
								Internal.Counter= 2
							else if(strcmp(adr(Internal.TmpDateTime),"Dec") = 0 )then
								Internal.DateTimeStruct.month= 12
								Internal.Counter= 2
							endif

						else if(Internal.Counter = 2) then
								Internal.DateTimeStruct.day= usint( atoi(adr(Internal.TmpDateTime)) )
								Internal.Counter= 3

						else if(Internal.Counter = 3) then
								Internal.DateTimeStruct.hour= usint( atoi(adr(Internal.TmpDateTime)) )
								Internal.Counter= 4

						else if(Internal.Counter = 4) then
								Internal.DateTimeStruct.minute= usint( atoi(adr(Internal.TmpDateTime)) )
								Internal.Counter= 5

						else if(Internal.Counter = 5) then
								Internal.DateTimeStruct.second= usint( atoi(adr(Internal.TmpDateTime)) )
								Internal.Counter= 6

						else if(Internal.Counter = 6) then
								Internal.DateTimeStruct.year= uint( atoi(adr(Internal.TmpDateTime)) )
								Internal.Counter= 7
						endif
						Internal.j= 0
					endif

				endloop
				Internal.i= 0
				Dyn_Date_and_Time access Internal.PV_Adress
				Dyn_Date_and_Time= DTStructure_TO_DT(adr(Internal.DateTimeStruct))
				Internal.DateAndTime = 0
				status= 65535
			else
				Internal.OnlyArrayInStruct = 0
				Internal.temp_status= DATATYP_ERROR
			endif

		else if( (strcmp(adr(Internal.DataTyp),"TIME") = 0 ) and (Internal.data_len = 4) and (Internal.PV_xgetadrStatus = 0) and (Internal.PV_nInfoStatus = 0) )then

			if (Internal.PVdata_typ = 12) then
				Dyn_Time access Internal.PV_Adress

				loop Internal.i=strlen(adr(Internal.Value)) downto 0 do	;Kommastellen löschen
					SearchChar access adr(Internal.Value)+Internal.i
					if(SearchChar ='.')then
						SearchChar= 0
						exitif(1=1)
					endif
				endloop
				Dyn_Time= time( atoi(adr(Internal.Value)) )
				status= 65535
			else
				Internal.OnlyArrayInStruct = 0
				Internal.temp_status= DATATYP_ERROR
			endif

		;######################################################################
		; keine DatentypKontrolle
		else if(No_DatatypControl = 1) and (Internal.PV_xgetadrStatus = 0) then
			; 1-Byte (BOOL,SINT,USINT)
			if (Internal.data_len = 1)	then
				Dyn_Usint access Internal.PV_Adress
				loop Internal.i=strlen(adr(Internal.Value)) downto 0 do	;Kommastellen löschen
					SearchChar access adr(Internal.Value)+Internal.i
					if(SearchChar ='.')then
						SearchChar= 0
						exitif(1=1)
					endif
				endloop
				Dyn_Usint= usint( atoi(adr(Internal.Value)) )
				status= 65535

			; 2-Byte (INT;UINT)
			else if (Internal.data_len = 2) and (Internal.PV_xgetadrStatus = 0) then
				Dyn_Uint access Internal.PV_Adress
				loop Internal.i=strlen(adr(Internal.Value)) downto 0 do	;Kommastellen löschen
					SearchChar access adr(Internal.Value)+Internal.i
					if(SearchChar ='.')then
						SearchChar= 0
						exitif(1=1)
					endif
				endloop
				Dyn_Uint= uint( atoi(adr(Internal.Value)) )
				status= 65535

			; 4-Byte (DINT,UDINT,TIME)
			else if (Internal.data_len = 4) and (Internal.DateAndTime = 0) and (Internal.PV_xgetadrStatus = 0) then
				Dyn_Udint access Internal.PV_Adress
				loop Internal.i=strlen(adr(Internal.Value)) downto 0 do	;Kommastellen löschen
					SearchChar access adr(Internal.Value)+Internal.i
					if(SearchChar ='.')then
						SearchChar= 0
						exitif(1=1)
					endif
				endloop
				Dyn_Udint= uint( atoi(adr(Internal.Value)) )
				status= 65535

			; 4-Byte (DATE_AND_TIME)
			else if (Internal.data_len = 4) and (Internal.DateAndTime = 1) and (Internal.PV_xgetadrStatus = 0) then
				Internal.Counter= 0
				loop Internal.i=0 to strlen(adr(Internal.DateTime)) do
					SearchChar access adr(Internal.DateTime)+Internal.i
					if( (SearchChar <> ' ') and (SearchChar <> ':') and (SearchChar <> 0) )then
						Internal.TmpDateTime[Internal.j]= SearchChar
						Internal.j= Internal.j+1
					else if( ((SearchChar = ' ') and (Internal.Counter < 3)) or ((SearchChar = ' ') and (Internal.Counter >= 5)) or ((SearchChar = ':') and (Internal.Counter >= 3)) or (SearchChar = 0) )then
						Internal.TmpDateTime[Internal.j]= 0
						; Tag
						if(Internal.Counter = 0) then
							if(strcmp(adr(Internal.TmpDateTime),"Sun") = 0 )then
								Internal.DateTimeStruct.wday= 0
								Internal.Counter = 1
							else if(strcmp(adr(Internal.TmpDateTime),"Mon") = 0 )then
								Internal.DateTimeStruct.wday= 1
								Internal.Counter = 1
							else if(strcmp(adr(Internal.TmpDateTime),"Tue") = 0 )then
								Internal.DateTimeStruct.wday= 2
								Internal.Counter = 1
							else if(strcmp(adr(Internal.TmpDateTime),"Wed") = 0 )then
								Internal.DateTimeStruct.wday= 3
								Internal.Counter = 1
							else if(strcmp(adr(Internal.TmpDateTime),"Thu") = 0 )then
								Internal.DateTimeStruct.wday= 4
								Internal.Counter = 1
							else if(strcmp(adr(Internal.TmpDateTime),"Fri") = 0 )then
								Internal.DateTimeStruct.wday= 5
								Internal.Counter = 1
							else if(strcmp(adr(Internal.TmpDateTime),"Sat") = 0 )then
								Internal.DateTimeStruct.wday= 6
								Internal.Counter = 1
							endif
						;Datum
						else if(Internal.Counter = 1) then
							if(strcmp(adr(Internal.TmpDateTime),"Jan") = 0 )then
								Internal.DateTimeStruct.month= 1
								Internal.Counter= 2
							else if(strcmp(adr(Internal.TmpDateTime),"Feb") = 0 )then
								Internal.DateTimeStruct.month= 2
								Internal.Counter= 2
							else if(strcmp(adr(Internal.TmpDateTime),"Mar") = 0 )then
								Internal.DateTimeStruct.month= 3
								Internal.Counter= 2
							else if(strcmp(adr(Internal.TmpDateTime),"Apr") = 0 )then
								Internal.DateTimeStruct.month= 4
								Internal.Counter= 2
							else if(strcmp(adr(Internal.TmpDateTime),"May") = 0 )then
								Internal.DateTimeStruct.month= 5
								Internal.Counter= 2
							else if(strcmp(adr(Internal.TmpDateTime),"Jun") = 0 )then
								Internal.DateTimeStruct.month= 6
								Internal.Counter= 2
							else if(strcmp(adr(Internal.TmpDateTime),"Jul") = 0 )then
								Internal.DateTimeStruct.month= 7
								Internal.Counter= 2
							else if(strcmp(adr(Internal.TmpDateTime),"Aug") = 0 )then
								Internal.DateTimeStruct.month= 8
								Internal.Counter= 2
							else if(strcmp(adr(Internal.TmpDateTime),"Sep") = 0 )then
								Internal.DateTimeStruct.month= 9
								Internal.Counter= 2
							else if(strcmp(adr(Internal.TmpDateTime),"Oct") = 0 )then
								Internal.DateTimeStruct.month= 10
								Internal.Counter= 2
							else if(strcmp(adr(Internal.TmpDateTime),"Nov") = 0 )then
								Internal.DateTimeStruct.month= 11
								Internal.Counter= 2
							else if(strcmp(adr(Internal.TmpDateTime),"Dec") = 0 )then
								Internal.DateTimeStruct.month= 12
								Internal.Counter= 2
							endif

						else if(Internal.Counter = 2) then
								Internal.DateTimeStruct.day= usint( atoi(adr(Internal.TmpDateTime)) )
								Internal.Counter= 3

						else if(Internal.Counter = 3) then
								Internal.DateTimeStruct.hour= usint( atoi(adr(Internal.TmpDateTime)) )
								Internal.Counter= 4

						else if(Internal.Counter = 4) then
								Internal.DateTimeStruct.minute= usint( atoi(adr(Internal.TmpDateTime)) )
								Internal.Counter= 5

						else if(Internal.Counter = 5) then
								Internal.DateTimeStruct.second= usint( atoi(adr(Internal.TmpDateTime)) )
								Internal.Counter= 6

						else if(Internal.Counter = 6) then
								Internal.DateTimeStruct.year= uint( atoi(adr(Internal.TmpDateTime)) )
								Internal.Counter= 7
						endif
						Internal.j= 0
					endif

				endloop
				Internal.i= 0
				Dyn_Date_and_Time access Internal.PV_Adress
				Dyn_Date_and_Time= DTStructure_TO_DT(adr(Internal.DateTimeStruct))
				Internal.DateAndTime = 0
				status= 65535

			; mehr als 4 Byte
			else if (Internal.data_len > 4) and (Internal.data_len <= sizeof(Dyn_String)) and (Internal.PV_xgetadrStatus = 0) then
				Dyn_String access Internal.PV_Adress
				strcpy(adr(Dyn_String),adr(Internal.Value))
				status= 65535
			else
				if(Internal.PV_xgetadrStatus <> 0)then
					Internal.OnlyArrayInStruct = 0
					Internal.temp_status= Internal.PV_xgetadrStatus
				else if (Internal.PV_nInfoStatus <> 0) then
					Internal.OnlyArrayInStruct = 0
					Internal.temp_status= Internal.PV_nInfoStatus
				else
					Internal.OnlyArrayInStruct = 0
					Internal.temp_status= DATATYP_ERROR
				endif
			endif

		; keine DatentypKontrolle
		;######################################################################
		else
				if(Internal.PV_xgetadrStatus <> 0)then
					Internal.OnlyArrayInStruct = 0
					Internal.temp_status= Internal.PV_xgetadrStatus
				else if (Internal.PV_nInfoStatus <> 0) then
					Internal.OnlyArrayInStruct = 0
					Internal.temp_status= Internal.PV_nInfoStatus
				else
					Internal.OnlyArrayInStruct = 0
					Internal.temp_status= DATATYP_ERROR
				endif
		endif

		when (Internal.Offset < FileOpen_CSV.filelen-1) and (status = 65535) and (Internal.temp_status = 0) do
			loop Internal.i=strlen(adr(Internal.StructName)) downto 0 do
				SearchChar access adr(Internal.StructName)+Internal.i
				if(SearchChar ='.')then
					SearchChar= 0
					exitif(1=1)
				endif
			endloop
			Internal.i= 0
			strcpy(adr(Internal.VarName),"")
		next SEARCH_VAR_NAMES

		when (Internal.Offset >= FileOpen_CSV.filelen-1) or (Internal.temp_status <> 0) do
		next TEMP_FREE

		;##########################################################################################
		state TEMP_FREE
		;##########################################################################################

			Internal.status_free= TMP_free(FileOpen_CSV.filelen,Internal.pFileData)

		when (1=1) do
			if(Internal.temp_status <> 0)then
				Internal.OnlyArrayInStruct = 0
				status= Internal.temp_status
			else if(Internal.status_free = 0)then
				Internal.OnlyArrayInStruct = 0
				status= 0
			else if(Internal.status_free <> 0)then
				Internal.OnlyArrayInStruct = 0
				status= Internal.status_free
			endif
			Internal.Step= 0
			exitif(1=1)
		next WAIT
	endselect

endloop
END_FUNCTION_BLOCK
```

#### ExListFile.ab
```automation-basic
FUNCTION_BLOCK ExListFile
;*****************************************************************
;FUB: 			ExFileList
;*****************************************************************
;Discription:
;	This FUB writes the Values from the allocated memory from the FUB
;	CSV-Init in a CSV-File.
;
;Parameter:
;
;Author:	Georg Kreil
;			B&R Eggelsberg
;
;History:	V0.01.1 - 24 June 2003
;					created
;			V0.01.2 - 8 July 2003
;					no changes
;			V0.01.3 - 14 July 2003
;					no changes
;			V0.01.4 - 15 July 2003
;					Error with maximum namelenght corrected
;					displayed strings changed by diplayed year
;					2003 -> 03
;					and without file-extension
;			V0.01.5 - 17 July 2003
;					no changes
;			V0.01.6 - 18 July 2003
;					Possibility to set the focus over a separate value added
;					Output, if it possible to scroll one page up/down  added
;			V0.01.7 - 7 August 2003
;					no changes
;			V0.01.8 - 8 August 2003
;					output strings one charecter shorter
;			V0.01.9 - 11 August 2003
;					no changes
;*****************************************************************

Internal.CRLF[0]= 13
Internal.CRLF[1]= 10
Internal.CRLF[2]= 0

	select Internal.Step

	;*********************************************************************
		state wait
	;*********************************************************************
	;*********************************************************************
	; control memorysize
    when ( (MaxNameLenght+19)*ArrayNum > SizeStringArray) or (MaxNameLenght > 28) do
    	status= MAX_NAMELENGHT_TO_LONG
    	command= 0
	next wait
	;*********************************************************************
	; create file-list
    when (command = FiJOB_CREATE_FILE_LIST ) and (status <> 65535) do
    	status  = 65535
		next file_dir_info
	;*********************************************************************
	; Scroll one line up
    when (command = FiJOB_LIST_UP) and (status <> 65535) do
	    	if(ListboxFocusPos = 0) then
	    		ListboxFocusPos= 0				; set focus
	        	ScrollUp= 0

	    		if (CSV_FileNum = 1) then ; set/reset scrolldown output
		        	ScrollDown= 0
	        	else
		        	ScrollDown= 1
	    		endif

	    	else
	    		ListboxFocusPos= ListboxFocusPos-1			; set focus

	    		if(ListboxFocusPos <> 0)then ;set/reset scrolldown output
		        	ScrollUp= 1
		        else
		        	ScrollUp= 0
		        endif

	    		if (CSV_FileNum = 1) then ; set/reset scrolldown output
		        	ScrollDown= 0
	        	else
		        	ScrollDown= 1
	    		endif

	    		if(Internal.DownLines < NumListboxLines-1)then
	    			Internal.UpLines= Internal.UpLines-1
	    			Internal.DownLines= Internal.DownLines+1
	    		else
	    			Internal.PosFirstLine= Internal.PosFirstLine-1
	    		endif
			endif
		command = 0
		status  = 0
		next wait
	;*********************************************************************
	; Scroll one line down
    when (command = FiJOB_LIST_DOWN) and (status <> 65535) do
	    	if(CSV_FileNum-1 <= ListboxFocusPos) then
	    		ListboxFocusPos= CSV_FileNum-1			; set focus
	    		ScrollDown= 0

	    		if (CSV_FileNum = 1) then ; set/reset scrollup output
		        	ScrollUp= 0
	        	else
		        	ScrollUp= 1
	    		endif

	    	else

	    		ListboxFocusPos= ListboxFocusPos+1			; set focus

	    		if(ListboxFocusPos <> CSV_FileNum-1 )then; set/reset scrollup output
		    		ScrollDown= 1
				else
		    		ScrollDown= 0
				endif

	    		if (CSV_FileNum = 1) then ; set/reset scrollup output
		        	ScrollUp= 0
	        	else
		        	ScrollUp= 1
	    		endif

	    		if(Internal.UpLines < NumListboxLines-1)then
	    			Internal.UpLines= Internal.UpLines+1
	    			Internal.DownLines= Internal.DownLines-1
	    		else
	    			Internal.PosFirstLine= Internal.PosFirstLine+1
	    		endif

			endif
		command = 0
		status  = 0
		next wait
	;*********************************************************************
	; Scroll one page up
    when (command = FiJOB_LIST_PG_UP) and (status <> 65535) do
	        ; there are less files as lines in the listbox
	    	if(ListboxFocusPos <= 0) or (ListboxFocusPos-NumListboxLines = 0)  then
	    		ListboxFocusPos= 0			; set focus
	        	ScrollUp= 0
    			Internal.UpLines= 0
    			Internal.DownLines= NumListboxLines-1
	    		Internal.PosFirstLine= 0

	    		if (CSV_FileNum = 1) then ; set/reset scrolldown output
		        	ScrollDown= 0
	        	else
		        	ScrollDown= 1
	    		endif

			else if ( ListboxFocusPos-NumListboxLines > 30000 )then
	        	ListboxFocusPos= 0			; set focus
	        	ScrollUp= 0
    			Internal.UpLines= 0
    			Internal.DownLines= NumListboxLines-1
	    		Internal.PosFirstLine= 0

	    		if (CSV_FileNum = 1) then ; set/reset scrolldown output
		        	ScrollDown= 0
	        	else
		        	ScrollDown= 1
	    		endif

			else if ( ListboxFocusPos-NumListboxLines > 0 )and ( ListboxFocusPos-NumListboxLines < 30000 )then
	        	ListboxFocusPos= ListboxFocusPos-NumListboxLines			; set focus
	        	ScrollUp= 1

	    		Internal.PosFirstLine= Internal.PosFirstLine - (NumListboxLines -Internal.UpLines)
    			Internal.UpLines= 0
    			Internal.DownLines= NumListboxLines-1

	    		if (CSV_FileNum = 1) then ; set/reset scrolldown output
		        	ScrollDown= 0
	        	else
		        	ScrollDown= 1
	    		endif

			endif
		command = 0
		status  = 0
		next wait
	;*********************************************************************
	; Scroll one page down
    when (command = FiJOB_LIST_PG_DOWN) and (status <> 65535) do
	        ; there are less files as lines in the listbox
	    	if(CSV_FileNum-1 <= ListboxFocusPos+NumListboxLines) then
	    		ListboxFocusPos= CSV_FileNum-1			; set focus
	    		ScrollDown= 0

    			if( CSV_FileNum > NumListboxLines) then
    				Internal.PosFirstLine= (CSV_FileNum-1)-(NumListboxLines-1)
   	 				Internal.UpLines= NumListboxLines-1
    				Internal.DownLines= 0
    			endif

	    		if (CSV_FileNum = 1) then ; set/reset scrollup output
		        	ScrollUp= 0
	        	else
		        	ScrollUp= 1
	    		endif

			else if ( ListboxFocusPos+NumListboxLines > CSV_FileNum )then
	        	ListboxFocusPos= CSV_FileNum-1			; set focus
	    		ScrollDown= 0

    			Internal.PosFirstLine= (CSV_FileNum-1)-(NumListboxLines-1)
    			Internal.UpLines= NumListboxLines-1
    			Internal.DownLines= 0

	    		if (CSV_FileNum = 1) then ; set/reset scrollup output
		        	ScrollUp= 0
	        	else
		        	ScrollUp= 1
	    		endif

			else if ( ListboxFocusPos+NumListboxLines < CSV_FileNum )then
	        	ListboxFocusPos= ListboxFocusPos+NumListboxLines			; set focus
	    		ScrollDown= 1

    			Internal.PosFirstLine= Internal.PosFirstLine + NumListboxLines - Internal.DownLines
    			Internal.UpLines= NumListboxLines-1
    			Internal.DownLines= 0

	    		if (CSV_FileNum = 1) then ; set/reset scrollup output
		        	ScrollUp= 0
	        	else
		        	ScrollUp= 1
	    		endif

			endif
		command = 0
		status  = 0
	    next wait

	;*********************************************************************
	; set focus with input-value
    when (command = FiJOB_SET_FOCUS) and (status <> 65535) do
  		if( SetFocusPos <= NumListboxLines-1  ) then
  			if( CSV_FileNum- 1 >= Internal.PosFirstLine+SetFocusPos ) then
		  		ListboxFocusPos= Internal.PosFirstLine+SetFocusPos
		  		Internal.DownLines= NumListboxLines-SetFocusPos-1
		  		Internal.UpLines= SetFocusPos
				status  = 0
			endif

		else
			status  = FOCUSPOS_OUT_OF_LISTBOX
		endif

	  	command = 0
   		next wait

	;*********************************************************************
		state file_dir_info
	;*********************************************************************

	  ; no memoryadress given
		when ( pStringArray = 0)  do
			command = 0
			status  = ERR_NO_MEM_ALLOC
		next wait

	    DirInfo_CSV.enable = 1
	    DirInfo_CSV.pDevice = pFileDevice
	    DirInfo_CSV.pPath = 0
	    DirInfo_CSV FUB DirInfo()

	    ;no error, files exists
	    when (DirInfo_CSV.status = ERRF_NO_ERROR) and (DirInfo_CSV.filenum <> 0) DO
	      Internal.FileNumOnDisk = uint(DirInfo_CSV.filenum)
	  	  memset(pStringArray, 0, SizeStringArray)
	      CSV_FileNum = 0								; filenumber reset
	      Internal.FileNumAct = 0                      	; actual filenumber reset
	      Internal.Offset = 0							; reset offset
	      status= 65535
		  strcpy(adr(Internal.TmpExtension),".CSV")
	      next file_info

	    ; no error, no files
	    when (DirInfo_CSV.status = ERRF_NO_ERROR) and (DirInfo_CSV.filenum = 0) DO
	      Internal.FileNumOnDisk = 0                    ; number of files reset
	      Internal.FileNumAct = 0                       ; actual filenumber reset
	      CSV_FileNum = 0								; filenumber reset
	   	  memset(pStringArray, 0,SizeStringArray)	  ; clear memory
	      command = 0  	                              ; command reset
	      status= 0  	      						  ; clear status
	      next wait

	    ; Fehler aufgetreten
	    when (DirInfo_CSV.status <> ERRF_NO_ERROR) and (DirInfo_CSV.status <> 65535) DO
	      status = DirInfo_CSV.status                  ; set error
	      command = 0                             	   ; command reset
	      Internal.FileNumAct = 0                      ; actual filenumber reset
	      Internal.Offset = 0      				       ; reset offset
	      next wait

	;*********************************************************************************
	  state file_info
	;*********************************************************************************

	    when (ArrayNum < Internal.FileNumOnDisk) DO
			command = 0
			status  = ARRAY_TO_LESS
    	next wait

	    ; create FileInfo
	    DirRead_CSV.enable = 1
	    DirRead_CSV.pDevice = pFileDevice
	    DirRead_CSV.pPath = 0
	    DirRead_CSV.entry = udint(Internal.FileNumAct)  ; actual filenumber
	    DirRead_CSV.option = FILE_FILE
	    DirRead_CSV.pData = adr(Internal.FileInfo)
	    DirRead_CSV.data_len = sizeof(Internal.FileInfo)
	    DirRead_CSV FUB DirRead()

	    ; Fehler aufgetreten
	    when (DirRead_CSV.status <> 0) and (DirRead_CSV.status <> 65535) do
	      status = DirRead_CSV.status                      ; Fehler setzen
	      command= 0
	      next wait

	    ; no error
	    if (DirRead_CSV.status = 0) then
	      ; filename to long -> not add to filelist
	      if (strlen(adr(Internal.FileInfo.Filename)) <= MaxNameLenght+4) then
			; control, if the file has the right extension
	      	loop Internal.i=0 to strlen(adr(Internal.FileInfo.Filename)) do
		     	memcpy(adr(Internal.TmpExtension),adr(Internal.FileInfo.Filename[Internal.i]),sizeof(Internal.TmpExtension))
		     	Internal.result1=strcmp(adr(Internal.TmpExtension),".CSV")
				Internal.result2=strcmp(adr(Internal.TmpExtension),".csv")

				; File gefunden
				if((Internal.result1 = 0 ) or (Internal.result2 = 0 ))then
					Internal.FileFound = 1
			    else if( adr(Internal.FileInfo.Filename[Internal.i]) = '.' )then
			    	exitif(1=1)			; File hat falsche Extension
			    endif

		    endloop

	      endif

	      Internal.FileNumAct = Internal.FileNumAct + 1                ;  increase actual filenumber
	    endif

		; ein neues CSV-File wurde gefunden
	    when(Internal.FileFound = 1) do
	    	Internal.FileFound = 0
	    	next open_file

	    when (Internal.FileNumAct >= Internal.FileNumOnDisk) DO		; all files listed
			command = 0								; reset command
			ListboxFocusPos= 0						; reset focus-position
	       	ScrollUp= 0
   			Internal.UpLines= 0
   			Internal.DownLines= NumListboxLines-1
   			Internal.PosFirstLine= 0

    		if (CSV_FileNum = 1) then
	        	ScrollDown= 0
        	else
	        	ScrollDown= 1
    		endif

			status  = 0		    					; reset status
      next wait

	;*********************************************************************************
	  state open_file
	;*********************************************************************************

		FileOpen_CSV.enable= 1
		FileOpen_CSV.pDevice= pFileDevice
		FileOpen_CSV.pFile= adr(Internal.FileInfo.Filename)
		FileOpen_CSV.mode= FILE_R
		FileOpen_CSV FUB FileOpen()

			; no error
			when (FileOpen_CSV.status = 0) do
				; allocate memory, to copy the first part of file
				Internal.status_alloc= TMP_alloc(FileOpen_CSV.filelen,adr(Internal.pFileData))
				status= 65535
			next read_file

			; file is opening
			when (FileOpen_CSV.status = 65535) do
				status= FileOpen_CSV.status
			next open_file

			;error durring opening
			when (FileOpen_CSV.status <> 0) and (FileOpen_CSV.status <> 65535) do
				status= FileOpen_CSV.status
			next wait

	;##########################################################################################
	state read_file
	;##########################################################################################

		if( (Internal.status_alloc = 0) and (FileOpen_CSV.status = 0) )then
			FileRead_CSV.enable= 1
			FileRead_CSV.ident= FileOpen_CSV.ident
			FileRead_CSV.offset= 0
			FileRead_CSV.pDest= Internal.pFileData
			FileRead_CSV.len= FileOpen_CSV.filelen
			FileRead_CSV FUB FileRead()
		endif

		; keine Speicher allokiert
		when (Internal.status_alloc <> 0) do
				status= Internal.status_alloc
			next wait

		; Fehler aufgetreten
		when (FileRead_CSV.status <> 0) and  (FileRead_CSV.status <> 65535) do
				status= FileRead_CSV.status
			next wait
		; noch beim Auslesen
		when (FileRead_CSV.status = 65535) do
				status= FileRead_CSV.status
			next read_file

		; fertig mit auslesen
		when (FileRead_CSV.status = 0) do
				status= 65535
			next close_file

		;##########################################################################################
		state close_file
		;##########################################################################################

		 	FileClose_CSV.enable= 1
			FileClose_CSV.ident= FileOpen_CSV.ident
			FileClose_CSV FUB FileClose()

			; Fehler beim Schliessen
			when (FileClose_CSV.status <> 0) and (FileClose_CSV.status <> 65535) do
				status= FileClose_CSV.status
			next wait

			; kein Fehler aufgetreten
			when (FileClose_CSV.status = 0) do
				status= 65535
			next search_filename

			; noch nicht fertig
			when (FileClose_CSV.status = 65535) do
				status= FileClose_CSV.status
			next close_file

		;##########################################################################################
		state search_filename
		;##########################################################################################

		; Kontrolle des Optionspointer
		when pOptions = 0 do
			status = ERR_ZERO_POINTER_OPTION
			next wait

		; Merker zurücksetzen
		Internal.PositionFound = 0
		Internal.FirstSeperatorFound = 0
		Internal.SecondSeperatorFound = 0
		Internal.EndPositionFound = 0

		; Optionsstruktur holen
		; -> kein Zeiger wegen debug-Möglichkeit
		memcpy( adr(Internal.OptionStruct), pOptions, sizeof(Internal.OptionStruct) )

		; ausgelesenes File durchsuchen
      	loop Internal.i=0 to Internal.OptionStruct.FileLenToRead do

      		; Position des Variablennamen im CSV-File suchen
			if (Internal.PositionFound = 0) then
				Internal.result1=memcmp( Internal.pFileData + Internal.i, adr(Internal.OptionStruct.SearchVarName), 5)
				if (Internal.result1 = 0) then
					Internal.PositionFound = 1	; Position gefunden
				endif
			; ersten ';' suchen
			else if (Internal.FirstSeperatorFound = 0 )then
				DynUsint access Internal.pFileData + Internal.i
				if (DynUsint = ';') then
					Internal.FirstSeperatorFound = 1 ; ersten ';' gefunden
				endif
			; zweiten ';' suchen
			else if (Internal.SecondSeperatorFound = 0 )then
				DynUsint access Internal.pFileData + Internal.i
				if (DynUsint = ';') then
					Internal.StartPositionName =  Internal.pFileData + Internal.i + 1 ;Startposition merken
					Internal.SecondSeperatorFound = 1 ; zweiten ';' gefunden
				endif
			; Ende der Zeile suchen
			else if (Internal.EndPositionFound = 0 )then
				DynUsint access Internal.pFileData + Internal.i
				if (DynUsint = 13) then
					; Variablenwert herauskopieren
					memcpy(adr(Internal.InternalFileName), Internal.StartPositionName, Internal.pFileData + Internal.i - Internal.StartPositionName);
					Internal.EndPositionFound = 1 ; Ende der Zeile gefunden
				endif
			endif
		endloop

		; Kompletten String löschen
		memset( adr(Internal.CompleteEntry), 0, sizeof(Internal.CompleteEntry) )
		;echten Filenamen "zusammenstutzen"
		memset( adr(Internal.FileInfo.Filename[strlen(adr(Internal.FileInfo.Filename)) - 4]), 0, sizeof(Internal.FileInfo.Filename)-strlen(adr(Internal.FileInfo.Filename))  )
		if ( strlen(adr(Internal.FileInfo.Filename)) > Internal.OptionStruct.MaxNrLen ) then
			Internal.FileInfo.Filename[Internal.OptionStruct.MaxNrLen] = 0
		else
			loop Internal.i = strlen(adr(Internal.FileInfo.Filename)) to Internal.OptionStruct.MaxNrLen-1 do
				Internal.FileInfo.Filename[Internal.i] = ' '
			endloop
		endif

		;echten Filenamen umkopieren
		memcpy( adr(Internal.CompleteEntry), adr(Internal.FileInfo.Filename) ,strlen(adr(Internal.FileInfo.Filename)) )
;		strcat( adr(Internal.CompleteEntry), "  ")

		;Filenamen "zusammenstutzen"
		if ( strlen(adr(Internal.InternalFileName)) > Internal.OptionStruct.MaxNameLen ) then
			Internal.InternalFileName[Internal.OptionStruct.MaxNameLen] = 0
		else
			loop Internal.i = strlen(adr(Internal.InternalFileName)) to Internal.OptionStruct.MaxNameLen-1 do
				Internal.InternalFileName[Internal.i] = ' '
			endloop
		endif
		;Filenamen hinzufügen zum echten Filenamen
		strcat( adr(Internal.CompleteEntry),adr(Internal.InternalFileName) )

		DT_TO_DTStructure(Internal.FileInfo.Date, adr(Internal.dateandtime));

		; create date and time to a string and add to the filename
		Internal.TmpString[0]= (Internal.dateandtime.day / 10) + '0'
		Internal.TmpString[1]= (Internal.dateandtime.day mod 10) + '0'
		Internal.TmpString[2]= '.'

		Internal.TmpString[3]= (Internal.dateandtime.month / 10) + '0'
		Internal.TmpString[4]= (Internal.dateandtime.month mod 10) + '0'
		Internal.TmpString[5]= '.'

		Internal.TmpString[6]= USINT( ((Internal.dateandtime.year mod 100)/10)  ) + '0'
		Internal.TmpString[7]= USINT(  (Internal.dateandtime.year mod 10)       ) + '0'
		Internal.TmpString[8]= ' '

		Internal.TmpString[9]= (Internal.dateandtime.hour / 10) + '0'
		Internal.TmpString[10]= (Internal.dateandtime.hour mod 10) + '0'
		Internal.TmpString[11]= ':'
		Internal.TmpString[12]= (Internal.dateandtime.minute / 10) + '0'
		Internal.TmpString[13]= (Internal.dateandtime.minute mod 10) + '0'
		Internal.TmpString[14]= 0

;		strcat( adr(Internal.CompleteEntry), " ")
		strcat( adr(Internal.CompleteEntry),adr(Internal.TmpString) )
		memset( adr(Internal.InternalFileName), 0, sizeof(Internal.InternalFileName) )

;		strcpy( pStringArray + Internal.Offset, adr(Internal.CompleteEntry) )
		strcpy( pStringArray + Internal.Offset, adr(Internal.CompleteEntry) )
		Internal.Offset = Internal.Offset + strlen( adr(Internal.CompleteEntry)) + 1

	    inc(CSV_FileNum)				; increase CSV-filenumber

	    when (Internal.FileNumAct >= Internal.FileNumOnDisk) DO		; all files listed
			command = 0								; reset command
			ListboxFocusPos= 0						; reset focus-position
	       	ScrollUp= 0
   			Internal.UpLines= 0
   			Internal.DownLines= NumListboxLines-1
   			Internal.PosFirstLine= 0

    		if (CSV_FileNum = 1) then
	        	ScrollDown= 0
        	else
	        	ScrollDown= 1
    		endif
			status  = 0		    					; reset status
    		next wait

		; nächster File holen
		when (1 = 1) do
			status= 65535
			next file_info

	endselect
END_FUNCTION_BLOCK
```

#### CSV_WriteFile.ab
```automation-basic
FUNCTION_BLOCK CSV_WriteFile
;*****************************************************************
;FUB: 			CSV_WriteFile
;*****************************************************************
;Discription:
;	This FUB writes the Values from the allocated memory from the FUB
;	CSV-Init in a CSV-File.
;
;Parameter:
;
;Author:	Georg Kreil
;			B&R Eggelsberg
;
;History:	V0.01 - 17 June 2003
;					created
;			V0.01.1 - 4 July 2003
;					no changes
;			V0.01.2 - 8 July 2003
;					no changes
;			V0.01.3 - 14 July 2003
;					no changes
;			V0.01.4 - 15 July 2003
;					no changes
;			V0.01.5 - 17 July 2003
;					no changes
;			V0.01.6 - 21 July 2003
;					no changes
;			V0.01.7 - 7 August 2003
;					no changes
;			V0.01.8 - 8 August 2003
;					no changes
;			V0.01.9 - 11 August 2003
;					no changes
;			V0.03   - 01 December 2003
;					underlines in filename allowed
;
;*****************************************************************

select Step

	;*************************************************************
	state CONTROL_FILENAME
	;*************************************************************

		when ( pFileName = 0) do
			status= ERROR_ZERO_POINTER_FILE
		next CONTROL_FILENAME

		strcpy(adr(FileName),pFileName)

		if( strlen(adr(FileName)) <> 0 )then
			; control, if the filename has the right extension
			loop i=0 to sizeof(FileName) do

				Dyn_Usint access (adr(FileName)+i)

				 if( ((Dyn_Usint >= '0' ) and ( Dyn_Usint <= '9' )) or ((Dyn_Usint >= 'A') and (Dyn_Usint <= 'Z')) or ((Dyn_Usint >= 'a') and (Dyn_Usint <= 'z')) or ( Dyn_Usint = '_') or ( Dyn_Usint = '-') or ( Dyn_Usint = '.') or ( Dyn_Usint = 0) )then

					if(Dyn_Usint = '.')then
						if ( strcmp((adr(FileName)+i),".CSV") = 0 ) or ( strcmp((adr(FileName)+i),".csv") = 0 ) then
							exitif(1=1)
						else
							strcpy((adr(FileName)+i),".CSV")
							exitif(1=1)
						endif
					else if(Dyn_Usint = 0) then
						strcpy((adr(FileName)+i),".CSV")
						exitif(1=1)
					endif
					status= 65535
				else
					status= INVALID_CHARACTER
					exitif(1=1)
				endif

			endloop

		;Pathname angegeben
		if(pPath <> 0)then
			strcpy(adr(Path),pPath)
			; Pathname bearbeiten
			if( strlen(adr(Path)) <> 0 )then

			; control, if the filename has the right extension
				loop i=0 to sizeof(Path) do

					Dyn_Usint access (adr(Path) + i)
					 if( ((Dyn_Usint >= '0' ) and ( Dyn_Usint <= '9' )) or ((Dyn_Usint >= 'A') and (Dyn_Usint <= 'Z')) or ((Dyn_Usint >= 'a') and (Dyn_Usint <= 'z')) or ( Dyn_Usint = '_') or ( Dyn_Usint = '-') or ( Dyn_Usint = '/') or ( Dyn_Usint = '\') or ( Dyn_Usint = 0) )then

						if(Dyn_Usint = 0) then
							Dyn_Usint access (adr(Path) + i - 1)
							if(Dyn_Usint <> '\') and (Dyn_Usint <> '/')then
								strcat( adr(Path), adr("/") )
							endif
							exitif(1=1)
						endif
						status= 65535
					else
						status= INVALID_CHARACTER
						exitif(1=1)
					endif
				endloop
				strcat( adr(Path), adr(FileName) )
				strcpy( adr(FileName), adr(Path) )
			endif
		endif

		else
			status= NO_FILENAME
		endif

		when ( pDevice = 0) do
			status= ERR_ZERO_POINTER_DEVICE
		next CONTROL_FILENAME

		when (status = 65535) do
		next CHECK_FILEDEVICE

	;*************************************************************
	state CHECK_FILEDEVICE
	;*************************************************************

		DirInfo_CSV.enable = 1
		DirInfo_CSV.pDevice = pDevice
		DirInfo_CSV.pPath = pPath
		DirInfo_CSV FUB DirInfo()

		; error
		when (DirInfo_CSV.status <> 0) and (DirInfo_CSV.status <> 65535) do
			status= DirInfo_CSV.status
		next CONTROL_FILENAME

		; no error
		when (DirInfo_CSV.status = 0) and ( (Mode = FILE_CREATE) or (Mode = FILE_OW)) do
			status= 65535
		next CHECK_PARTITION

		when (DirInfo_CSV.status = 0) and ( (Mode = FILE_CREATE_WITHOUT_MEM_CHECK) or (Mode = FILE_OW_WITHOUT_MEM_CHECK)) do
			status= 65535
		next FILE_CREATE

		; file is under creation
		when (DirInfo_CSV.status = 65535) do
			status= DirInfo_CSV.status
		next CHECK_FILEDEVICE

	;*************************************************************
	state CHECK_PARTITION
	;*************************************************************

		DevMemInfo_CSV.enable= 1
		DevMemInfo_CSV.pDevice= pDevice
		DevMemInfo_CSV FUB DevMemInfo()
		; error
		when (DevMemInfo_CSV.status <> 0) and (DevMemInfo_CSV.status <> 65535) do
			status= DevMemInfo_CSV.status
		next CONTROL_FILENAME

		; no error, enough memory
		when (DevMemInfo_CSV.status = 0) and (DevMemInfo_CSV.freemem >= MemLen ) do
			status= 65535
		next FILE_CREATE

		; no error, not enough memory
		when (DevMemInfo_CSV.status = 0) and (DevMemInfo_CSV.freemem < MemLen ) do
			status= fiERR_SPACE
		next CONTROL_FILENAME

		; file is under creation
		when (DevMemInfo_CSV.status = 65535) do
			status= DevMemInfo_CSV.status
		next CHECK_PARTITION

	;*************************************************************
	state FILE_CREATE
	;*************************************************************

		FileCreate_CSV.enable= 1
		FileCreate_CSV.pDevice= pDevice
		FileCreate_CSV.pFile= adr(FileName)
		FileCreate_CSV FUB FileCreate()

		; file allready exists and will be not overwritten
		when (FileCreate_CSV.status = 20705) and (Mode <> FILE_OW) and (Mode <> FILE_OW_WITHOUT_MEM_CHECK) do
			status= FileCreate_CSV.status
		next  CONTROL_FILENAME

		; file allready exists and will be overwritten
		when (FileCreate_CSV.status = 20705) and ( (Mode = FILE_OW) or (Mode = FILE_OW_WITHOUT_MEM_CHECK) ) do
			status= 65535
		next FILE_DELETE

		; error
		when (FileCreate_CSV.status <> 0) and (FileCreate_CSV.status <> 65535) do
			status= FileCreate_CSV.status
		next CONTROL_FILENAME

		; no error
		when (FileCreate_CSV.status = 0) do
			FileWrite_CSV.ident= FileCreate_CSV.ident
			status= 65535
		next FILE_WRITE

		; file is under creation
		when (FileCreate_CSV.status = 65535) do
			status= FileCreate_CSV.status
		next FILE_CREATE

	;*************************************************************
	state FILE_DELETE
	;*************************************************************
		FileDelete_CSV.enable= 1
		FileDelete_CSV.pDevice= pDevice
		FileDelete_CSV.pName= adr(FileName)
		FileDelete_CSV FUB FileDelete()

		; error
		when (FileDelete_CSV.status <> 0) and (FileDelete_CSV.status <> 65535) do
			status= FileDelete_CSV.status
		next CONTROL_FILENAME

		; no error
		when (FileDelete_CSV.status = 0) do
			status= 65535
		next FILE_CREATE

		; file under erasing
		when (FileDelete_CSV.status = 65535) do
			status= FileDelete_CSV.status
		next FILE_DELETE

	;*************************************************************
	state FILE_WRITE
	;*************************************************************

		FileWrite_CSV.enable= 1
		FileWrite_CSV.offset= 0
		FileWrite_CSV.pSrc= pStructMem
		FileWrite_CSV.len= MemLen
		FileWrite_CSV FUB FileWrite()

		; error
		when (FileWrite_CSV.status <> 0) and (FileWrite_CSV.status <> 65535) do
			status= FileWrite_CSV.status
		next CONTROL_FILENAME

		; no error
		when (FileWrite_CSV.status = 0) do
			status= 65535
		next FILE_CLOSE

		; file is writeing
		when (FileWrite_CSV.status = 65535) do
			status= FileWrite_CSV.status
		next FILE_WRITE

	;*************************************************************
	state FILE_CLOSE
	;*************************************************************

		FileClose_CSV.enable= 1
		FileClose_CSV.ident= FileWrite_CSV.ident
		FileClose_CSV FUB FileClose()

		; error
		when (FileClose_CSV.status <> 0) and (FileClose_CSV.status <> 65535) do
			status= FileClose_CSV.status
		next CONTROL_FILENAME

		; no error
		when (FileClose_CSV.status = 0) do
			status= 0
		next CONTROL_FILENAME

		; file is closing
		when (FileClose_CSV.status = 65535) do
			status= FileClose_CSV.status
		next FILE_CLOSE

endselect
END_FUNCTION_BLOCK
```

#### CSV_AtoDouble.ab - Converts an ASCII-String to a LREAL-Value
```automation-basic
(********************************************************************
 * COPYRIGHT -- Bernecker + Rainer
 ********************************************************************
 * Library: CSV_File
 * File: CSV_AtoDouble.ab
 * Author: diermayrd
 * Created: August 10, 2010
 ********************************************************************
 * Implementation of library CSV_File
 ********************************************************************)

(* Converts an ASCII-String to a LREAL-Value *)
FUNCTION CSV_AtoDouble

	;get Lenght of the String
	intStrLeng	= strlen(pString)

	if (intStrLeng > 0) then
		;String is not empty -> start of conversion
		;------------------------------------------

		;==========================================
		;check if value is negative -> search "-"
		;==========================================

		;reset String which would be used to conversion and copy Symbol
		memset(adr(tempString),0,sizeof(tempString))
		memcpy(adr(tempString),pString,sizeof(tempString))

		if (tempString = '-') then
			;Value is negativ
			negativeValue		= TRUE
			startIndexIntPart	= 1
		else
			;Value is positiv
			negativeValue		= FALSE
			startIndexIntPart	= 0
		endif

		;==========================================
		;convert Integer Part
		;==========================================

		;reset internal Values
		lRealIntegerPart	= 0
		startIndexDecPart	= 0
		anzExponent			= 0
		decimalPlaces		= FALSE

		loop i=startIndexIntPart to (intStrLeng-1) do

			;reset String which would be used to conversion and copy Symbol
			memset(adr(tempString),0,sizeof(tempString))
			memcpy(adr(tempString),pString+i,sizeof(tempString))

			if ( (tempString = 'e') or (tempString = 'E') ) then
				;start of Exponent -> copy Value
				;-----------------------------------
				;sign
				memset(adr(tempString),0,sizeof(tempString))
				memcpy(adr(tempString),pString+i+1,sizeof(tempString))
				if (tempString = '-') then
					;negativ
					positivExponent	= FALSE
					;exponent
					anzExponent	= atoi(pString+i+2)
					exitif(1=1)
				else
					;positiv
					positivExponent	= TRUE
					;exponent
					anzExponent	= atoi(pString+i+1)
					exitif(1=1)
				endif
				;-----------------------------------

			else if ((tempString = '.') or (tempString = ',')) then
				;Decimalpoint found -> end of Integer Part
				;exit loop;
				decimalPlaces		= TRUE
				startIndexDecPart	= i+1
				exitif (1=1)
			else
				;convert AscII to Integer
				tempInt	= atoi(adr(tempString))
				;convert Inteegr to LREAL and add to lRealIntPart
				lRealIntegerPart	= lRealIntegerPart*10+lreal(tempInt)
			endif

		endloop

		;==========================================
		;convert Decimal Part
		;==========================================

		;reset internal Values
		lRealDecimalPart	= 0
		anzDecimalPlaces	= 0

		if (decimalPlaces = TRUE) then
			;Decimal Places existing -> start conversion
			anzExponent	= 0

			loop i=startIndexDecPart to (intStrLeng-1) do

				;reset String which would be used to conversion and copy Symbol
				memset(adr(tempString),0,sizeof(tempString))
				memcpy(adr(tempString),pString+i,sizeof(tempString))

				if ( (tempString = 'e') or (tempString = 'E') ) then
					;start of Exponent -> copy Value
					;-----------------------------------
					;sign
					memset(adr(tempString),0,sizeof(tempString))
					memcpy(adr(tempString),pString+i+1,sizeof(tempString))
					if (tempString = '-') then
						;negativ
						positivExponent	= FALSE
						;exponent
						anzExponent	= atoi(pString+i+2)
						exitif(1=1)
					else
						;positiv
						positivExponent	= TRUE
						;exponent
						anzExponent	= atoi(pString+i+1)
						exitif(1=1)
					endif
					;-----------------------------------

				else
					;convert AscII to Integer
					tempInt	= atoi(adr(tempString))
					;convert Inteegr to LREAL and add to lRealIntPart
					lRealDecimalPart	= lRealDecimalPart*10+lreal(tempInt)
					anzDecimalPlaces	= anzDecimalPlaces+1
				endif

			endloop

			;divide Value to get from 456123 -> 0.456123
			;-------------------------------------------
			loop i=1 to anzDecimalPlaces do
				;divide by 10;
				lRealDecimalPart	= lRealDecimalPart/10
			endloop
		else
			lRealDecimalPart	= 0.0
		endif

		;==========================================
		;add Integer Part and Decimal Part
		;==========================================

		if (negativeValue = TRUE) then
			;Value is negativ -> muliplicate with (-1)
			CSV_AtoDouble = (lRealIntegerPart+lRealDecimalPart)*(-1)
		else
			;Value is positiv
			CSV_AtoDouble	= lRealIntegerPart+lRealDecimalPart
		endif

		;==========================================
		;calculate exponential-faktor
		;==========================================

		if (positivExponent = TRUE) then
			;multiplie Value
			;-------------------------------------------
			loop i=1 to uint(anzExponent) do
				;multiplie by 10;
				CSV_AtoDouble	= CSV_AtoDouble*10
			endloop
		else
			;divide Value
			;-------------------------------------------
			loop i=1 to uint(anzExponent) do
				;divide by 10;
				CSV_AtoDouble	= CSV_AtoDouble/10
			endloop
		endif

	else
		;String is empty -> write 0.0 to value
		;------------------------------------------
		CSV_AtoDouble	= 0.0
	endif

END_FUNCTION
```

#### CSV_DoubleToA.ab - Function to convert a LREAL-Value to an ASCII-String
```automation-basic
(********************************************************************
 * COPYRIGHT -- Bernecker + Rainer
 ********************************************************************
 * Library: CSV_File
 * File: CSV_DoubleToA.ab
 * Author: diermayrd
 * Created: August 12, 2010
 ********************************************************************
 * Implementation of library CSV_File
 ********************************************************************)

(* Function to convert a LREAL-Value to an ASCII-String *)
FUNCTION CSV_DoubleToA

;copy lReal-Value to temp Variable
tempLREALvalue	= lRealValue
intStringLen	= strlen(pString)
memset(pString,0,intStringLen)

if (tempLREALvalue <> 0.0) then

	;==========================================
	;check value of sign
	;==========================================

	tempInt	= 0
	memcpy(adr(tempInt),adr(tempLREALvalue)+7,sizeof(tempInt))
	negativeValue	= bit_tst(tempInt,7) ;highest BIT is for sign

	if (negativeValue = TRUE) then
		;multiple value with *(-1) -> to get positiv value
		tempLREALvalue	= tempLREALvalue*(-1)
	endif

	;==========================================
	;get exponent and sign of exponent
	;==========================================

	if (tempLREALvalue < 1.0) then
		;Value smaller than 1 -> multiplicate Value till bigger than 1
		loop i=1 to 400 do
			;Exponent can be maximal 380 -> loop till 400 because before 400 will be EXIT
			tempLREALvalue	= tempLREALvalue*10

			if (tempLREALvalue >= 1.0) then
				;Value in correct Range -> save exponent + get IntPart + EXIT loop
				exponent		= i*(-1)
				IntPartLReal	= trunc(tempLREALvalue)
				exitif(1=1)
			endif
		endloop

	else if (tempLREALvalue >= 10.0) then
		;Value bigger or equal 10 -> divide Value till smaller than 10
		loop i=1 to 400 do
			;Exponent can be maximal 380 -> loop till 400 because before 400 will be EXIT
			tempLREALvalue	= tempLREALvalue/10

			if (tempLREALvalue < 10.0) then
				;Value in correct Range -> save exponent + get IntPart + EXIT loop
				exponent		= i
				IntPartLReal	= trunc(tempLREALvalue)
				exitif(1=1)
			endif
		endloop
	else
		;Value in range 1 <= value < 10
		exponent		= 0
		IntPartLReal	= trunc(tempLREALvalue)
	endif

	;==========================================
	;get decimal part
	;==========================================

	;detach calculated decimal part and multiplie with 10 to get next decimal Part
	;1.2345 -> 0.2345 -> 2.345 -> //  and so on
	tempLREALvalue	= tempLREALvalue-lreal(IntPartLReal)
	tempLREALvalue	= tempLREALvalue*10
	;reset decimalPart-Array
	memset(adr(DecPartLReal),0,sizeof(DecPartLReal))

	loop i=0 to 13 do
		;maximum 14 decimal places accuracy for LREAL
		DecPartLReal[i]	= trunc(tempLREALvalue)

		;detach calculated decimal part and multiplie with 10 to get next decimal Part
		;1.2345 -> 0.2345 -> 2.345 -> //  and so on
		tempLREALvalue	= tempLREALvalue-lreal(DecPartLReal[i])
		tempLREALvalue	= tempLREALvalue*10
	endloop

	;==========================================
	;create String with all components
	;==========================================

	;sign
	;------------------------------------------
	if (negativeValue = TRUE) then
		;write "-"
		strcpy(pString,"-")
	endif

	;Integer Part
	;------------------------------------------
	memset(adr(tempString),0,sizeof(tempString))
	itoa(IntPartLReal,adr(tempString))
	if (negativeValue = TRUE) then
		strcat(pString,adr(tempString))
	else
		strcpy(pString,adr(tempString))
	endif

	;"."
	;------------------------------------------
	strcat(pString,".")

	;Decimal Places
	;------------------------------------------
	firstEntry	= FALSE
	memset(adr(tempDecString),0,sizeof(tempDecString))

	loop i=13 downto 0 do
		exitif(i<0)
		memset(adr(tempString),0,sizeof(tempString))
		itoa(DecPartLReal[i],adr(tempString))
		if ((DecPartLReal[i] = 0) and (firstEntry = FALSE) ) then
			;when decimalpart is 0 and it will be the first entry -> don't write it
		else
			if (firstEntry = FALSE) then
				;first write process to string -> strcpy instead of strcat
				strcpy(adr(tempDecString),adr(tempString))
				firstEntry	= TRUE
			else
				strcat(adr(tempDecString),adr(tempString))
			endif
		endif
	endloop

	;swop content of Decimal Places
	intStringLen	= strlen(adr(tempDecString))
	memset(adr(tempString),0,sizeof(tempString))

	if (intStringLen > 0) then
		intStringLen	= intStringLen-1
		loop i=0 to intStringLen do
		memcpy((adr(tempString)+i),(adr(tempDecString)+(intStringLen-i)),1)
		endloop
	else
		strcpy(adr(tempString),"0");
	endif
	strcat(pString,adr(tempString))

	;"e"
	;------------------------------------------
	strcat(pString,"e")

	;sign of exponent
	;------------------------------------------
	if (exponent >= 0) then
		;positiv -> add + befor exponent
		strcat(pString,"+")
	endif

	;exponent
	;------------------------------------------
	memset(adr(tempString),0,sizeof(tempString))
	itoa(exponent,adr(tempString))
	strcat(pString,adr(tempString))

else
	strcpy(pString,"0.0")
endif

CSV_DoubleToA = strlen(pString)

END_FUNCTION
```

### Library Logical/Libraries/HlpStr (IEC, version 1.00.0)
Depends on: standard, AsBrStr, AsBrMath

#### HlpStr.fun - Exported functions and function blocks
```iecst
(********************************************************************
 * COPYRIGHT -- Bernecker + Rainer
 ********************************************************************
 * Library: HlpStr
 * File: HlpStr.fun
 * Author: beutert
 * Created: May 21, 2010
 ********************************************************************
 * Functions and function blocks of library HlpStr
 ********************************************************************)

FUNCTION findstr : UINT (*find a specified string in a given string*)
	VAR_INPUT
		IN1 : STRING[1000];
		IN2 : STRING[80];
		StartPos : UINT;
	END_VAR
	VAR
		ReturnVal : UINT;
		Str2 : STRING[1000];
		wStrLen : UINT;
	END_VAR
END_FUNCTION

FUNCTION_BLOCK findchar (*find a specified character in a given string*)
	VAR_INPUT
		enable : BOOL;
		pString : UDINT;
		Char : USINT;
		StartPos : UINT;
	END_VAR
	VAR_OUTPUT
		CharPos : UINT;
		status : UINT;
	END_VAR
	VAR
		ptByte_a : REFERENCE TO ARRAY[0..999] OF USINT;
		wStrLen : UINT;
		CharFound : BOOL;
	END_VAR
END_FUNCTION_BLOCK

FUNCTION LTRIM : UINT (*delete blanks at beginning of string*)
	VAR_INPUT
		enable : BOOL;
		pString : UDINT;
	END_VAR
	VAR
		status : UINT;
		szHlpStr1 : STRING[1000];
		wStrLen : UINT;
		pByte : REFERENCE TO USINT;
		wStrLenHlp : UINT;
	END_VAR
END_FUNCTION

FUNCTION l2str : UINT (*convert an UDINT value to string*)
	VAR_INPUT
		value : UDINT;
		pString : UDINT;
	END_VAR
	VAR
		lRest : UDINT;
		ii : USINT;
		lDivisor : UDINT;
		lQuot : UDINT;
		szQuot : STRING[80];
	END_VAR
END_FUNCTION

FUNCTION RTRIM : UINT (*TODO: Add your comment here*)
	VAR_INPUT
		enable : BOOL;
		pString : UDINT;
	END_VAR
	VAR
		status : UINT;
		szHlpStr1 : STRING[1000];
		wStrLen : UINT;
		pByte : REFERENCE TO USINT;
		wStrLenHlp : UINT;
		bDbg : USINT;
	END_VAR
END_FUNCTION

FUNCTION TRIM : UINT (*TODO: Add your comment here*)
	VAR_INPUT
		enable : BOOL;
		pString : UDINT;
	END_VAR
	VAR
		status : UINT;
	END_VAR
END_FUNCTION
```

#### findstr.ab
```automation-basic
(********************************************************************
 * COPYRIGHT -- Bernecker + Rainer
 ********************************************************************
 * Library: HlpStr
 * File: findstr.ab
 * Author: beutert
 * Created: May 21, 2010
 ********************************************************************
 * Implementation of library HlpStr
 ********************************************************************
 Function: find a specified string in a given string

    input:  string (STRING[1000])
            search string (STRING[80])
            starting position (UINT)
   output:  position of string (UINT)
 ********************************************************************)

FUNCTION findstr
	wStrLen = UINT(brsstrlen(adr(IN1)));		//length of string to be searched

	if ((StartPos = 0) or (StartPos > wStrLen)) then
		ReturnVal = 0;	//no starting position (=0) specified or starting position > length of string
	else
	Str2 = MID(IN1, wStrLen, StartPos);			//copy part of string starting from starting position
	ReturnVal = FIND(Str2, IN2);						//and then search for string (IN2)
	if (ReturnVal <> 0) then
		ReturnVal = ReturnVal + StartPos - 1;	//if string is found, calculate position in original string
	endif;
  endif;
	findstr = ReturnVal;

END_FUNCTION
```

#### findchar.ab
```automation-basic
(********************************************************************
 * COPYRIGHT -- Microsoft
 ********************************************************************
 * Library: HlpStr
 * File: findchar.ab
 * Author: beutert
 * Created: March 25, 2011
 ********************************************************************
 * Implementation of library HlpStr
 ********************************************************************
 Function: find a specified character in a given string

    input:  enable (BOOL)
						pointer to string (UDINT)
            character (USINT)
            starting position (UINT)
   output:  position of character in string (UINT)
            status (UINT)
 ********************************************************************)

FUNCTION_BLOCK findchar

	if (enable = true) then
		ptByte_a access pString;
		wStrLen = UINT(brsstrlen(pString));
	  CharPos = 0;

		if (wStrLen > UINT(sizeof(ptByte_a))) then
			status = 50000;	//string too long
		else if ((StartPos > wStrLen) or (StartPos = 0)) then
			status = 50001;	//starting position invalid
		else
			status = 65535;	//busy
			CharFound = false;
			loop CharPos = StartPos-1 to wStrLen - 1 do
				if (ptByte_a[CharPos] = Char) then
					CharPos = CharPos + 1;
					CharFound = true;
					status = 0;	//everything fine
					exitif (1=1);
				endif;
			endloop;
			if (CharFound = false) then
				CharPos = 0;
				status = 50002;	//character not found
			endif;
		endif;	//wStrLen > UINT(sizeof(ptByte_a))
	else
		status = 65534;
	endif;	//enable = true

END_FUNCTION_BLOCK
```

#### LTRIM.ab
```automation-basic
(********************************************************************
 * COPYRIGHT -- Microsoft
 ********************************************************************
 * Library: HlpStr
 * File: LTRIM.ab
 * Author: beutert
 * Created: March 25, 2011
 ********************************************************************
 * Implementation of library HlpStr
 ********************************************************************
 Function: delete blanks at beginning of string

    input:  pointer to string (UDINT)
   output:  status
 ********************************************************************)

FUNCTION LTRIM
	if (enable = true) then
		wStrLenHlp = UINT(sizeof(szHlpStr1) - 1);
		wStrLen = UINT(brsstrlen(pString));
		if (wStrLen > wStrLenHlp) then
			status = 50000;	//string too long
		else
			status = 65535;
			brsstrcpy(adr(szHlpStr1),pString);
			loop
				pByte access adr(szHlpStr1);
				if (pByte = ' ') then
					szHlpStr1 = RIGHT(szHlpStr1, INT(wStrLen) - 1);
					wStrLen = wStrLen - 1;
				else
					exitif (1=1);
				endif;
			endloop;
			brsstrcpy(pString,adr(szHlpStr1));
			status = 0;
		endif;
	else
		status = 65534;
	endif;
	LTRIM = status;
END_FUNCTION
```
